LIN {X 0,Y 438.796,Z 820.121,A -85,B 0,C 180,E1 6106.016,E2 6106.016} C_VEL
LIN {X 0,Y 435.592,Z 843.834,A -85,B 0,C 180,E1 6105.62,E2 6105.62} C_VEL
LIN {X 0,Y 431.491,Z 865.928,A -85,B 0,C 180,E1 6105.195,E2 6105.195} C_VEL
LIN {X 0,Y 425.589,Z 891.228,A -85,B 0,C 180,E1 6104.584,E2 6104.584} C_VEL
LIN {X 0,Y 418.146,Z 916.547,A -85,B 0,C 180,E1 6103.788,E2 6103.788} C_VEL
LIN {X 0,Y 411.227,Z 936.788,A -85,B 0,C 180,E1 6103.015,E2 6103.015} C_VEL
LIN {X 0,Y 403.474,Z 956.852,A -85,B 0,C 180,E1 6102.103,E2 6102.103} C_VEL
LIN {X 0,Y 393.277,Z 980.389,A -85,B 0,C 180,E1 6100.823,E2 6100.823} C_VEL
LIN {X 0,Y 381.687,Z 1003.698,A -85,B 0,C 180,E1 6099.261,E2 6099.261} C_VEL
LIN {X 0,Y 371.951,Z 1021.583,A -85,B 0,C 180,E1 6097.831,E2 6097.831} C_VEL
LIN {X 0,Y 361.684,Z 1038.996,A -85,B 0,C 180,E1 6096.212,E2 6096.212} C_VEL
LIN {X 0,Y 348.484,Z 1059.817,A -85,B 0,C 180,E1 6093.904,E2 6093.904} C_VEL
LIN {X 0,Y 335.22,Z 1078.877,A -85,B 0,C 180,E1 6091.299,E2 6091.299} C_VEL
LIN {X 0,Y 323.717,Z 1094.534,A -85,B 0,C 180,E1 6088.74,E2 6088.74} C_VEL
LIN {X 0,Y 310.823,Z 1111.367,A -85,B 0,C 180,E1 6085.438,E2 6085.438} C_VEL
LIN {X 0,Y 298.275,Z 1126.865,A -85,B 0,C 180,E1 6081.666,E2 6081.666} C_VEL
LIN {X 0,Y 288.449,Z 1138.762,A -85,B 0,C 180,E1 6078.182,E2 6078.182} C_VEL
LIN {X 0,Y 279.204,Z 1149.91,A -85,B 0,C 180,E1 6074.292,E2 6074.292} C_VEL
LIN {X 0,Y 269.366,Z 1162.072,A -85,B 0,C 180,E1 6069.121,E2 6069.121} C_VEL
LIN {X 0,Y 261.736,Z 1171.778,A -85,B 0,C 180,E1 6063.899,E2 6063.899} C_VEL
LIN {X 0,Y 256.571,Z 1179.002,A -85,B 0,C 180,E1 6059.152,E2 6059.152} C_VEL
LIN {X 0,Y 252.751,Z 1185.047,A -85,B 0,C 180,E1 6054.294,E2 6054.294} C_VEL
LIN {X 0,Y 249.904,Z 1190.603,A -85,B 0,C 180,E1 6048.667,E2 6048.667} C_VEL
LIN {X 0,Y 248.427,Z 1194.755,A -85,B 0,C 180,E1 6042.789,E2 6042.789} C_VEL
LIN {X 0,Y 248.033,Z 1197.119,A -85,B 0,C 180,E1 6037.644,E2 6037.644} C_VEL
LIN {X 0,Y 247.993,Z 1198.227,A -85,B 0,C 180,E1 6033.235,E2 6033.235} C_VEL
LIN {X 0,Y 248.003,Z 1198.443,A -85,B 0,C 180,E1 6028.844,E2 6028.844} C_VEL
LIN {X 0,Y 247.993,Z 1197.691,A -85,B 0,C 180,E1 6024.214,E2 6024.214} C_VEL
LIN {X 0,Y 248.182,Z 1195.889,A -85,B 0,C 180,E1 6019.435,E2 6019.435} C_VEL
LIN {X 0,Y 248.942,Z 1193.015,A -85,B 0,C 180,E1 6014.575,E2 6014.575} C_VEL
LIN {X 0,Y 250.577,Z 1189.058,A -85,B 0,C 180,E1 6009.686,E2 6009.686} C_VEL
LIN {X 0,Y 253.211,Z 1184.216,A -85,B 0,C 180,E1 6005.006,E2 6005.006} C_VEL
LIN {X 0,Y 257.322,Z 1177.869,A -85,B 0,C 180,E1 6000.058,E2 6000.058} C_VEL
LIN {X 0,Y 264.391,Z 1168.312,A -85,B 0,C 180,E1 5994.113,E2 5994.113} C_VEL
LIN {X 0,Y 272.385,Z 1158.147,A -85,B 0,C 180,E1 5989.131,E2 5989.131} C_VEL
LIN {X 0,Y 280.522,Z 1148.247,A -85,B 0,C 180,E1 5985.11,E2 5985.11} C_VEL
LIN {X 0,Y 290.427,Z 1136.32,A -85,B 0,C 180,E1 5981.064,E2 5981.064} C_VEL
LIN {X 0,Y 303.233,Z 1120.644,A -85,B 0,C 180,E1 5976.748,E2 5976.748} C_VEL
LIN {X 0,Y 314.417,Z 1106.504,A -85,B 0,C 180,E1 5973.572,E2 5973.572} C_VEL
LIN {X 0,Y 325.807,Z 1091.588,A -85,B 0,C 180,E1 5970.762,E2 5970.762} C_VEL
LIN {X 0,Y 339.632,Z 1072.555,A -85,B 0,C 180,E1 5967.788,E2 5967.788} C_VEL
LIN {X 0,Y 352.367,Z 1053.518,A -85,B 0,C 180,E1 5965.371,E2 5965.371} C_VEL
LIN {X 0,Y 363.194,Z 1036.239,A -85,B 0,C 180,E1 5963.528,E2 5963.528} C_VEL
LIN {X 0,Y 374.64,Z 1016.568,A -85,B 0,C 180,E1 5961.754,E2 5961.754} C_VEL
LIN {X 0,Y 386.839,Z 993.292,A -85,B 0,C 180,E1 5960.023,E2 5960.023} C_VEL
LIN {X 0,Y 396.09,Z 973.641,A -85,B 0,C 180,E1 5958.801,E2 5958.801} C_VEL
LIN {X 0,Y 404.283,Z 954.413,A -85,B 0,C 180,E1 5957.788,E2 5957.788} C_VEL
LIN {X 0,Y 412.183,Z 933.675,A -85,B 0,C 180,E1 5956.866,E2 5956.866} C_VEL
LIN {X 0,Y 421.033,Z 906.617,A -85,B 0,C 180,E1 5955.886,E2 5955.886} C_VEL
LIN {X 0,Y 427.259,Z 883.572,A -85,B 0,C 180,E1 5955.226,E2 5955.226} C_VEL
LIN {X 0,Y 432.073,Z 862.129,A -85,B 0,C 180,E1 5954.733,E2 5954.733} C_VEL
LIN {X 0,Y 436.664,Z 836.034,A -85,B 0,C 180,E1 5954.249,E2 5954.249} C_VEL
LIN {X 0,Y 441.088,Z 795.407,A -85,B 0,C 180,E1 5953.614,E2 5953.614} C_VEL
LIN {X 0,Y 460.609,Z 598.366,A -85,B 0,C 180,E1 5950.681,E2 5950.681} C_VEL
LIN {X 0,Y 457.6,Z 592.689,A -85,B 0,C 180,E1 5948.418,E2 5948.418} C_VEL
LIN {X 0,Y 455.635,Z 589.003,A -85,B 0,C 180,E1 5946.616,E2 5946.616} C_VEL
LIN {X 0,Y 454.128,Z 586.275,A -85,B 0,C 180,E1 5944.926,E2 5944.926} C_VEL
LIN {X 0,Y 452.252,Z 582.816,A -85,B 0,C 180,E1 5941.901,E2 5941.901} C_VEL
LIN {X 0,Y 451.266,Z 582.034,A -85,B 0,C 180,E1 5938.222,E2 5938.222} C_VEL
LIN {X 0,Y 451.505,Z 582.728,A -85,B 0,C 180,E1 5935.682,E2 5935.682} C_VEL
LIN {X 0,Y 453.105,Z 586.957,A -85,B 0,C 180,E1 5931.945,E2 5931.945} C_VEL
LIN {X 0,Y 454.885,Z 591.279,A -85,B 0,C 180,E1 5929.616,E2 5929.616} C_VEL
LIN {X 0,Y 457.288,Z 596.631,A -85,B 0,C 180,E1 5927.306,E2 5927.306} C_VEL
LIN {X 0,Y 459.279,Z 601.556,A -85,B 0,C 180,E1 5925.696,E2 5925.696} C_VEL
LIN {X 0,Y 437.308,Z 826.32,A -85,B 0,C 180,E1 5922.449,E2 5922.449} C_VEL
LIN {X 0,Y 434.141,Z 848.783,A -85,B 0,C 180,E1 5922.078,E2 5922.078} C_VEL
LIN {X 0,Y 428.807,Z 875.909,A -85,B 0,C 180,E1 5921.533,E2 5921.533} C_VEL
LIN {X 0,Y 422.894,Z 898.914,A -85,B 0,C 180,E1 5920.937,E2 5920.937} C_VEL
LIN {X 0,Y 416.442,Z 920.116,A -85,B 0,C 180,E1 5920.253,E2 5920.253} C_VEL
LIN {X 0,Y 408.237,Z 943.42,A -85,B 0,C 180,E1 5919.329,E2 5919.329} C_VEL
LIN {X 0,Y 398.118,Z 967.799,A -85,B 0,C 180,E1 5918.126,E2 5918.126} C_VEL
LIN {X 0,Y 389.491,Z 986.265,A -85,B 0,C 180,E1 5917.032,E2 5917.032} C_VEL
LIN {X 0,Y 379.607,Z 1005.443,A -85,B 0,C 180,E1 5915.694,E2 5915.694} C_VEL
LIN {X 0,Y 366.696,Z 1028.066,A -85,B 0,C 180,E1 5913.779,E2 5913.779} C_VEL
LIN {X 0,Y 355.286,Z 1046.089,A -85,B 0,C 180,E1 5911.919,E2 5911.919} C_VEL
LIN {X 0,Y 344.633,Z 1061.765,A -85,B 0,C 180,E1 5910.001,E2 5910.001} C_VEL
LIN {X 0,Y 332.718,Z 1078.203,A -85,B 0,C 180,E1 5907.614,E2 5907.614} C_VEL
LIN {X 0,Y 318.568,Z 1096.284,A -85,B 0,C 180,E1 5904.382,E2 5904.382} C_VEL
LIN {X 0,Y 307.782,Z 1109.336,A -85,B 0,C 180,E1 5901.53,E2 5901.53} C_VEL
LIN {X 0,Y 297.229,Z 1121.639,A -85,B 0,C 180,E1 5898.315,E2 5898.315} C_VEL
LIN {X 0,Y 284.778,Z 1135.724,A -85,B 0,C 180,E1 5893.764,E2 5893.764} C_VEL
LIN {X 0,Y 275.658,Z 1145.826,A -85,B 0,C 180,E1 5889.673,E2 5889.673} C_VEL
LIN {X 0,Y 268.203,Z 1154.193,A -85,B 0,C 180,E1 5885.562,E2 5885.562} C_VEL
LIN {X 0,Y 260.633,Z 1163.104,A -85,B 0,C 180,E1 5880.17,E2 5880.17} C_VEL
LIN {X 0,Y 254.816,Z 1170.36,A -85,B 0,C 180,E1 5874.332,E2 5874.332} C_VEL
LIN {X 0,Y 251.596,Z 1175.02,A -85,B 0,C 180,E1 5869.502,E2 5869.502} C_VEL
LIN {X 0,Y 249.485,Z 1178.756,A -85,B 0,C 180,E1 5864.388,E2 5864.388} C_VEL
LIN {X 0,Y 248.338,Z 1181.722,A -85,B 0,C 180,E1 5858.335,E2 5858.335} C_VEL
LIN {X 0,Y 248.049,Z 1182.949,A -85,B 0,C 180,E1 5853.004,E2 5853.004} C_VEL
LIN {X 0,Y 248.038,Z 1183.109,A -85,B 0,C 180,E1 5848.615,E2 5848.615} C_VEL
LIN {X 0,Y 248.144,Z 1182.396,A -85,B 0,C 180,E1 5843.987,E2 5843.987} C_VEL
LIN {X 0,Y 248.625,Z 1180.776,A -85,B 0,C 180,E1 5839.34,E2 5839.34} C_VEL
LIN {X 0,Y 249.756,Z 1178.231,A -85,B 0,C 180,E1 5834.68,E2 5834.68} C_VEL
LIN {X 0,Y 251.931,Z 1174.534,A -85,B 0,C 180,E1 5829.801,E2 5829.801} C_VEL
LIN {X 0,Y 256.315,Z 1168.527,A -85,B 0,C 180,E1 5823.845,E2 5823.845} C_VEL
LIN {X 0,Y 262.455,Z 1160.894,A -85,B 0,C 180,E1 5818.283,E2 5818.283} C_VEL
LIN {X 0,Y 269.126,Z 1153.218,A -85,B 0,C 180,E1 5813.792,E2 5813.792} C_VEL
LIN {X 0,Y 278.439,Z 1142.928,A -85,B 0,C 180,E1 5808.917,E2 5808.917} C_VEL
LIN {X 0,Y 289.405,Z 1130.604,A -85,B 0,C 180,E1 5804.343,E2 5804.343} C_VEL
LIN {X 0,Y 299.489,Z 1119.152,A -85,B 0,C 180,E1 5800.873,E2 5800.873} C_VEL
LIN {X 0,Y 311.744,Z 1104.868,A -85,B 0,C 180,E1 5797.305,E2 5797.305} C_VEL
LIN {X 0,Y 324.711,Z 1088.751,A -85,B 0,C 180,E1 5794.074,E2 5794.074} C_VEL
LIN {X 0,Y 335.895,Z 1074.082,A -85,B 0,C 180,E1 5791.642,E2 5791.642} C_VEL
LIN {X 0,Y 346.923,Z 1058.74,A -85,B 0,C 180,E1 5789.495,E2 5789.495} C_VEL
LIN {X 0,Y 360.604,Z 1038.215,A -85,B 0,C 180,E1 5787.12,E2 5787.12} C_VEL
LIN {X 0,Y 371.794,Z 1019.69,A -85,B 0,C 180,E1 5785.364,E2 5785.364} C_VEL
LIN {X 0,Y 381.756,Z 1001.755,A -85,B 0,C 180,E1 5783.925,E2 5783.925} C_VEL
LIN {X 0,Y 392.363,Z 980.824,A -85,B 0,C 180,E1 5782.517,E2 5782.517} C_VEL
LIN {X 0,Y 403.186,Z 956.416,A -85,B 0,C 180,E1 5781.18,E2 5781.18} C_VEL
LIN {X 0,Y 410.938,Z 936.563,A -85,B 0,C 180,E1 5780.286,E2 5780.286} C_VEL
LIN {X 0,Y 417.942,Z 916.134,A -85,B 0,C 180,E1 5779.508,E2 5779.508} C_VEL
LIN {X 0,Y 425.586,Z 889.88,A -85,B 0,C 180,E1 5778.706,E2 5778.706} C_VEL
LIN {X 0,Y 431.196,Z 865.565,A -85,B 0,C 180,E1 5778.142,E2 5778.142} C_VEL
LIN {X 0,Y 435.188,Z 843.579,A -85,B 0,C 180,E1 5777.734,E2 5777.734} C_VEL
LIN {X 0,Y 436.959,Z 831.119,A -85,B 0,C 180,E1 5777.528,E2 5777.528} C_VEL
LIN {X 0,Y 437.578,Z 823.596,A -85,B 0,C 180,E1 5777.288,E2 5777.288} C_VEL
LIN {X 0,Y 437.97,Z 804.029,A -85,B 0,C 180,E1 5776.203,E2 5776.203} C_VEL
LIN {X 0,Y 438.401,Z 797.543,A -85,B 0,C 180,E1 5776.014,E2 5776.014} C_VEL
LIN {X 0,Y 457.292,Z 607.146,A -85,B 0,C 180,E1 5773.293,E2 5773.293} C_VEL
LIN {X 0,Y 454.572,Z 600.576,A -85,B 0,C 180,E1 5770.776,E2 5770.776} C_VEL
LIN {X 0,Y 452.457,Z 595.594,A -85,B 0,C 180,E1 5768.131,E2 5768.131} C_VEL
LIN {X 0,Y 451.655,Z 593.668,A -85,B 0,C 180,E1 5766.738,E2 5766.738} C_VEL
LIN {X 0,Y 450.659,Z 590.496,A -85,B 0,C 180,E1 5763.434,E2 5763.434} C_VEL
LIN {X 0,Y 450.86,Z 590.358,A -85,B 0,C 180,E1 5759.873,E2 5759.873} C_VEL
LIN {X 0,Y 451.639,Z 591.215,A -85,B 0,C 180,E1 5757.843,E2 5757.843} C_VEL
LIN {X 0,Y 453.942,Z 595.56,A -85,B 0,C 180,E1 5754.375,E2 5754.375} C_VEL
LIN {X 0,Y 456.023,Z 599.584,A -85,B 0,C 180,E1 5752.25,E2 5752.25} C_VEL
LIN {X 0,Y 458.505,Z 604.367,A -85,B 0,C 180,E1 5750.218,E2 5750.218} C_VEL
LIN {X 0,Y 436.503,Z 821.567,A -85,B 0,C 180,E1 5747.007,E2 5747.007} C_VEL
LIN {X 0,Y 433.318,Z 844.483,A -85,B 0,C 180,E1 5746.628,E2 5746.628} C_VEL
LIN {X 0,Y 429.076,Z 866.856,A -85,B 0,C 180,E1 5746.203,E2 5746.203} C_VEL
LIN {X 0,Y 422.777,Z 893.065,A -85,B 0,C 180,E1 5745.574,E2 5745.574} C_VEL
LIN {X 0,Y 415.449,Z 917.389,A -85,B 0,C 180,E1 5744.817,E2 5744.817} C_VEL
LIN {X 0,Y 408.62,Z 937.002,A -85,B 0,C 180,E1 5744.081,E2 5744.081} C_VEL
LIN {X 0,Y 400.598,Z 957.382,A -85,B 0,C 180,E1 5743.17,E2 5743.17} C_VEL
LIN {X 0,Y 389.823,Z 981.671,A -85,B 0,C 180,E1 5741.862,E2 5741.862} C_VEL
LIN {X 0,Y 378.65,Z 1003.647,A -85,B 0,C 180,E1 5740.405,E2 5740.405} C_VEL
LIN {X 0,Y 368.503,Z 1021.888,A -85,B 0,C 180,E1 5738.969,E2 5738.969} C_VEL
LIN {X 0,Y 357.598,Z 1039.945,A -85,B 0,C 180,E1 5737.302,E2 5737.302} C_VEL
LIN {X 0,Y 343.413,Z 1061.561,A -85,B 0,C 180,E1 5734.89,E2 5734.89} C_VEL
LIN {X 0,Y 331.214,Z 1078.635,A -85,B 0,C 180,E1 5732.564,E2 5732.564} C_VEL
LIN {X 0,Y 319.585,Z 1094.023,A -85,B 0,C 180,E1 5730.07,E2 5730.07} C_VEL
LIN {X 0,Y 306.717,Z 1110.28,A -85,B 0,C 180,E1 5726.908,E2 5726.908} C_VEL
LIN {X 0,Y 293.101,Z 1126.583,A -85,B 0,C 180,E1 5722.964,E2 5722.964} C_VEL
LIN {X 0,Y 282.726,Z 1138.66,A -85,B 0,C 180,E1 5719.403,E2 5719.403} C_VEL
LIN {X 0,Y 273.221,Z 1149.634,A -85,B 0,C 180,E1 5715.529,E2 5715.529} C_VEL
LIN {X 0,Y 262.87,Z 1161.797,A -85,B 0,C 180,E1 5710.287,E2 5710.287} C_VEL
LIN {X 0,Y 254.667,Z 1171.673,A -85,B 0,C 180,E1 5704.856,E2 5704.856} C_VEL
LIN {X 0,Y 249.292,Z 1178.739,A -85,B 0,C 180,E1 5700.089,E2 5700.089} C_VEL
LIN {X 0,Y 245.19,Z 1184.787,A -85,B 0,C 180,E1 5695.094,E2 5695.094} C_VEL
LIN {X 0,Y 242.112,Z 1190.347,A -85,B 0,C 180,E1 5689.292,E2 5689.292} C_VEL
LIN {X 0,Y 240.489,Z 1194.504,A -85,B 0,C 180,E1 5683.218,E2 5683.218} C_VEL
LIN {X 0,Y 240.04,Z 1196.87,A -85,B 0,C 180,E1 5677.9,E2 5677.9} C_VEL
LIN {X 0,Y 239.994,Z 1197.98,A -85,B 0,C 180,E1 5673.343,E2 5673.343} C_VEL
LIN {X 0,Y 240.006,Z 1198.196,A -85,B 0,C 180,E1 5668.806,E2 5668.806} C_VEL
LIN {X 0,Y 239.997,Z 1197.442,A -85,B 0,C 180,E1 5664.021,E2 5664.021} C_VEL
LIN {X 0,Y 240.199,Z 1195.698,A -85,B 0,C 180,E1 5659.203,E2 5659.203} C_VEL
LIN {X 0,Y 241.043,Z 1192.797,A -85,B 0,C 180,E1 5654.11,E2 5654.11} C_VEL
LIN {X 0,Y 242.841,Z 1188.8,A -85,B 0,C 180,E1 5649.009,E2 5649.009} C_VEL
LIN {X 0,Y 245.692,Z 1183.955,A -85,B 0,C 180,E1 5644.185,E2 5644.185} C_VEL
LIN {X 0,Y 249.987,Z 1177.748,A -85,B 0,C 180,E1 5639.205,E2 5639.205} C_VEL
LIN {X 0,Y 257.286,Z 1168.461,A -85,B 0,C 180,E1 5633.238,E2 5633.238} C_VEL
LIN {X 0,Y 265.956,Z 1157.992,A -85,B 0,C 180,E1 5627.994,E2 5627.994} C_VEL
LIN {X 0,Y 274.595,Z 1147.97,A -85,B 0,C 180,E1 5623.865,E2 5623.865} C_VEL
LIN {X 0,Y 284.932,Z 1136.038,A -85,B 0,C 180,E1 5619.779,E2 5619.779} C_VEL
LIN {X 0,Y 298.25,Z 1120.349,A -85,B 0,C 180,E1 5615.446,E2 5615.446} C_VEL
LIN {X 0,Y 309.832,Z 1106.204,A -85,B 0,C 180,E1 5612.272,E2 5612.272} C_VEL
LIN {X 0,Y 320.911,Z 1092.143,A -85,B 0,C 180,E1 5609.623,E2 5609.623} C_VEL
LIN {X 0,Y 334.737,Z 1073.742,A -85,B 0,C 180,E1 5606.73,E2 5606.73} C_VEL
LIN {X 0,Y 348.221,Z 1054.156,A -85,B 0,C 180,E1 5604.244,E2 5604.244} C_VEL
LIN {X 0,Y 359.322,Z 1036.885,A -85,B 0,C 180,E1 5602.41,E2 5602.41} C_VEL
LIN {X 0,Y 370.456,Z 1018.221,A -85,B 0,C 180,E1 5600.736,E2 5600.736} C_VEL
LIN {X 0,Y 383.154,Z 994.751,A -85,B 0,C 180,E1 5598.989,E2 5598.989} C_VEL
LIN {X 0,Y 392.996,Z 974.303,A -85,B 0,C 180,E1 5597.729,E2 5597.729} C_VEL
LIN {X 0,Y 401.43,Z 954.907,A -85,B 0,C 180,E1 5596.722,E2 5596.722} C_VEL
LIN {X 0,Y 409.456,Z 934.239,A -85,B 0,C 180,E1 5595.817,E2 5595.817} C_VEL
LIN {X 0,Y 418.228,Z 908.105,A -85,B 0,C 180,E1 5594.881,E2 5594.881} C_VEL
LIN {X 0,Y 424.87,Z 883.989,A -85,B 0,C 180,E1 5594.2,E2 5594.2} C_VEL
LIN {X 0,Y 429.753,Z 862.607,A -85,B 0,C 180,E1 5593.717,E2 5593.717} C_VEL
LIN {X 0,Y 434.19,Z 837.948,A -85,B 0,C 180,E1 5593.265,E2 5593.265} C_VEL
LIN {X 0,Y 438.389,Z 801.607,A -85,B 0,C 180,E1 5592.697,E2 5592.697} C_VEL
LIN {X 0,Y 458.297,Z 604.189,A -85,B 0,C 180,E1 5589.782,E2 5589.782} C_VEL
LIN {X 0,Y 455.023,Z 597.759,A -85,B 0,C 180,E1 5587.005,E2 5587.005} C_VEL
LIN {X 0,Y 453.034,Z 594.148,A -85,B 0,C 180,E1 5584.811,E2 5584.811} C_VEL
LIN {X 0,Y 451.209,Z 590.714,A -85,B 0,C 180,E1 5581.778,E2 5581.778} C_VEL
LIN {X 0,Y 450.286,Z 589.974,A -85,B 0,C 180,E1 5578.218,E2 5578.218} C_VEL
LIN {X 0,Y 450.525,Z 590.758,A -85,B 0,C 180,E1 5575.672,E2 5575.672} C_VEL
LIN {X 0,Y 452.006,Z 594.767,A -85,B 0,C 180,E1 5572.117,E2 5572.117} C_VEL
LIN {X 0,Y 453.731,Z 599.105,A -85,B 0,C 180,E1 5569.782,E2 5569.782} C_VEL
LIN {X 0,Y 456.149,Z 604.706,A -85,B 0,C 180,E1 5567.402,E2 5567.402} C_VEL
LIN {X 0,Y 457.073,Z 607.226,A -85,B 0,C 180,E1 5566.599,E2 5566.599} C_VEL
LIN {X 0,Y 435.048,Z 827.651,A -85,B 0,C 180,E1 5563.446,E2 5563.446} C_VEL
LIN {X 0,Y 431.48,Z 851.887,A -85,B 0,C 180,E1 5563.048,E2 5563.048} C_VEL
LIN {X 0,Y 425.687,Z 879.45,A -85,B 0,C 180,E1 5562.485,E2 5562.485} C_VEL
LIN {X 0,Y 420.148,Z 900.383,A -85,B 0,C 180,E1 5561.942,E2 5561.942} C_VEL
LIN {X 0,Y 413.814,Z 920.754,A -85,B 0,C 180,E1 5561.294,E2 5561.294} C_VEL
LIN {X 0,Y 405.067,Z 945.091,A -85,B 0,C 180,E1 5560.34,E2 5560.34} C_VEL
LIN {X 0,Y 395.195,Z 968.26,A -85,B 0,C 180,E1 5559.207,E2 5559.207} C_VEL
LIN {X 0,Y 386.266,Z 986.989,A -85,B 0,C 180,E1 5558.114,E2 5558.114} C_VEL
LIN {X 0,Y 375.96,Z 1006.562,A -85,B 0,C 180,E1 5556.762,E2 5556.762} C_VEL
LIN {X 0,Y 362.417,Z 1029.615,A -85,B 0,C 180,E1 5554.814,E2 5554.814} C_VEL
LIN {X 0,Y 351.157,Z 1046.969,A -85,B 0,C 180,E1 5553.029,E2 5553.029} C_VEL
LIN {X 0,Y 339.838,Z 1063.18,A -85,B 0,C 180,E1 5551.047,E2 5551.047} C_VEL
LIN {X 0,Y 325.684,Z 1082.015,A -85,B 0,C 180,E1 5548.257,E2 5548.257} C_VEL
LIN {X 0,Y 313.213,Z 1097.329,A -85,B 0,C 180,E1 5545.449,E2 5545.449} C_VEL
LIN {X 0,Y 302.128,Z 1110.305,A -85,B 0,C 180,E1 5542.587,E2 5542.587} C_VEL
LIN {X 0,Y 290.168,Z 1123.778,A -85,B 0,C 180,E1 5538.995,E2 5538.995} C_VEL
LIN {X 0,Y 277.901,Z 1136.994,A -85,B 0,C 180,E1 5534.556,E2 5534.556} C_VEL
LIN {X 0,Y 268.925,Z 1146.538,A -85,B 0,C 180,E1 5530.592,E2 5530.592} C_VEL
LIN {X 0,Y 260.812,Z 1155.24,A -85,B 0,C 180,E1 5526.185,E2 5526.185} C_VEL
LIN {X 0,Y 252.439,Z 1164.551,A -85,B 0,C 180,E1 5520.201,E2 5520.201} C_VEL
LIN {X 0,Y 247.16,Z 1170.861,A -85,B 0,C 180,E1 5514.881,E2 5514.881} C_VEL
LIN {X 0,Y 243.774,Z 1175.472,A -85,B 0,C 180,E1 5509.904,E2 5509.904} C_VEL
LIN {X 0,Y 241.45,Z 1179.371,A -85,B 0,C 180,E1 5504.294,E2 5504.294} C_VEL
LIN {X 0,Y 240.319,Z 1182.098,A -85,B 0,C 180,E1 5498.133,E2 5498.133} C_VEL
LIN {X 0,Y 240.054,Z 1183.196,A -85,B 0,C 180,E1 5493.104,E2 5493.104} C_VEL
LIN {X 0,Y 240.041,Z 1183.356,A -85,B 0,C 180,E1 5488.568,E2 5488.568} C_VEL
LIN {X 0,Y 240.16,Z 1182.644,A -85,B 0,C 180,E1 5483.786,E2 5483.786} C_VEL
LIN {X 0,Y 240.647,Z 1181.134,A -85,B 0,C 180,E1 5479.224,E2 5479.224} C_VEL
LIN {X 0,Y 241.919,Z 1178.482,A -85,B 0,C 180,E1 5474.171,E2 5474.171} C_VEL
LIN {X 0,Y 244.264,Z 1174.786,A -85,B 0,C 180,E1 5469.138,E2 5469.138} C_VEL
LIN {X 0,Y 248.838,Z 1168.92,A -85,B 0,C 180,E1 5463.132,E2 5463.132} C_VEL
LIN {X 0,Y 255.488,Z 1161.128,A -85,B 0,C 180,E1 5457.292,E2 5457.292} C_VEL
LIN {X 0,Y 262.5,Z 1153.477,A -85,B 0,C 180,E1 5452.726,E2 5452.726} C_VEL
LIN {X 0,Y 271.811,Z 1143.635,A -85,B 0,C 180,E1 5447.972,E2 5447.972} C_VEL
LIN {X 0,Y 283.18,Z 1131.432,A -85,B 0,C 180,E1 5443.335,E2 5443.335} C_VEL
LIN {X 0,Y 293.876,Z 1119.731,A -85,B 0,C 180,E1 5439.742,E2 5439.742} C_VEL
LIN {X 0,Y 304.982,Z 1107.202,A -85,B 0,C 180,E1 5436.561,E2 5436.561} C_VEL
LIN {X 0,Y 319.647,Z 1089.718,A -85,B 0,C 180,E1 5432.976,E2 5432.976} C_VEL
LIN {X 0,Y 330.981,Z 1075.293,A -85,B 0,C 180,E1 5430.575,E2 5430.575} C_VEL
LIN {X 0,Y 341.93,Z 1060.496,A -85,B 0,C 180,E1 5428.494,E2 5428.494} C_VEL
LIN {X 0,Y 353.969,Z 1043.092,A -85,B 0,C 180,E1 5426.435,E2 5426.435} C_VEL
LIN {X 0,Y 367.623,Z 1021.367,A -85,B 0,C 180,E1 5424.337,E2 5424.337} C_VEL
LIN {X 0,Y 377.967,Z 1003.21,A -85,B 0,C 180,E1 5422.885,E2 5422.885} C_VEL
LIN {X 0,Y 387.734,Z 984.447,A -85,B 0,C 180,E1 5421.621,E2 5421.621} C_VEL
LIN {X 0,Y 398.725,Z 960.887,A -85,B 0,C 180,E1 5420.304,E2 5420.304} C_VEL
LIN {X 0,Y 407.816,Z 938.233,A -85,B 0,C 180,E1 5419.277,E2 5419.277} C_VEL
LIN {X 0,Y 414.921,Z 918.031,A -85,B 0,C 180,E1 5418.513,E2 5418.513} C_VEL
LIN {X 0,Y 421.939,Z 894.911,A -85,B 0,C 180,E1 5417.8,E2 5417.8} C_VEL
LIN {X 0,Y 428.578,Z 867.625,A -85,B 0,C 180,E1 5417.156,E2 5417.156} C_VEL
LIN {X 0,Y 432.761,Z 845.353,A -85,B 0,C 180,E1 5416.743,E2 5416.743} C_VEL
LIN {X 0,Y 435.945,Z 821.931,A -85,B 0,C 180,E1 5416.369,E2 5416.369} C_VEL
LIN {X 0,Y 438.401,Z 797.543,A -85,B 0,C 180,E1 5416.014,E2 5416.014} C_VEL
LIN {X 0,Y 438.892,Z 790.003,A -85,B 0,C 180,E1 5415.78,E2 5415.78} C_VEL
LIN {X 0,Y 439.359,Z 770.428,A -85,B 0,C 180,E1 5414.702,E2 5414.702} C_VEL
LIN {X 0,Y 439.841,Z 763.942,A -85,B 0,C 180,E1 5414.516,E2 5414.516} C_VEL
LIN {X 0,Y 455.199,Z 612.867,A -85,B 0,C 180,E1 5412.383,E2 5412.383} C_VEL
LIN {X 0,Y 452.836,Z 607.181,A -85,B 0,C 180,E1 5409.982,E2 5409.982} C_VEL
LIN {X 0,Y 451.17,Z 602.87,A -85,B 0,C 180,E1 5407.641,E2 5407.641} C_VEL
LIN {X 0,Y 450.237,Z 600.725,A -85,B 0,C 180,E1 5405.787,E2 5405.787} C_VEL
LIN {X 0,Y 449.679,Z 598.441,A -85,B 0,C 180,E1 5403.442,E2 5403.442} C_VEL
LIN {X 0,Y 449.878,Z 598.3,A -85,B 0,C 180,E1 5399.873,E2 5399.873} C_VEL
LIN {X 0,Y 450.647,Z 599.257,A -85,B 0,C 180,E1 5397.838,E2 5397.838} C_VEL
LIN {X 0,Y 452.779,Z 603.355,A -85,B 0,C 180,E1 5394.551,E2 5394.551} C_VEL
LIN {X 0,Y 454.74,Z 607.263,A -85,B 0,C 180,E1 5392.482,E2 5392.482} C_VEL
LIN {X 0,Y 456.293,Z 610.506,A -85,B 0,C 180,E1 5391.114,E2 5391.114} C_VEL
LIN {X 0,Y 434.186,Z 824.271,A -85,B 0,C 180,E1 5387.988,E2 5387.988} C_VEL
LIN {X 0,Y 430.933,Z 846.6,A -85,B 0,C 180,E1 5387.621,E2 5387.621} C_VEL
LIN {X 0,Y 425.667,Z 873.141,A -85,B 0,C 180,E1 5387.114,E2 5387.114} C_VEL
LIN {X 0,Y 419.035,Z 898.394,A -85,B 0,C 180,E1 5386.476,E2 5386.476} C_VEL
LIN {X 0,Y 412.514,Z 919.346,A -85,B 0,C 180,E1 5385.822,E2 5385.822} C_VEL
LIN {X 0,Y 405.159,Z 939.866,A -85,B 0,C 180,E1 5385.052,E2 5385.052} C_VEL
LIN {X 0,Y 395.344,Z 963.949,A -85,B 0,C 180,E1 5383.959,E2 5383.959} C_VEL
LIN {X 0,Y 384.408,Z 987.004,A -85,B 0,C 180,E1 5382.667,E2 5382.667} C_VEL
LIN {X 0,Y 374.507,Z 1005.884,A -85,B 0,C 180,E1 5381.404,E2 5381.404} C_VEL
LIN {X 0,Y 364.006,Z 1024.227,A -85,B 0,C 180,E1 5379.955,E2 5379.955} C_VEL
LIN {X 0,Y 350.636,Z 1045.616,A -85,B 0,C 180,E1 5377.936,E2 5377.936} C_VEL
LIN {X 0,Y 337.702,Z 1064.338,A -85,B 0,C 180,E1 5375.773,E2 5375.773} C_VEL
LIN {X 0,Y 325.994,Z 1080.211,A -85,B 0,C 180,E1 5373.586,E2 5373.586} C_VEL
LIN {X 0,Y 313.862,Z 1095.753,A -85,B 0,C 180,E1 5371.037,E2 5371.037} C_VEL
LIN {X 0,Y 298.393,Z 1114.433,A -85,B 0,C 180,E1 5367.252,E2 5367.252} C_VEL
LIN {X 0,Y 286.736,Z 1127.81,A -85,B 0,C 180,E1 5363.891,E2 5363.891} C_VEL
LIN {X 0,Y 276.389,Z 1139.387,A -85,B 0,C 180,E1 5360.403,E2 5360.403} C_VEL
LIN {X 0,Y 265.024,Z 1152.015,A -85,B 0,C 180,E1 5355.793,E2 5355.793} C_VEL
LIN {X 0,Y 254.412,Z 1163.785,A -85,B 0,C 180,E1 5350.318,E2 5350.318} C_VEL
LIN {X 0,Y 247.32,Z 1171.984,A -85,B 0,C 180,E1 5345.603,E2 5345.603} C_VEL
LIN {X 0,Y 241.582,Z 1179.133,A -85,B 0,C 180,E1 5340.582,E2 5340.582} C_VEL
LIN {X 0,Y 236.537,Z 1186.386,A -85,B 0,C 180,E1 5334.206,E2 5334.206} C_VEL
LIN {X 0,Y 233.536,Z 1191.719,A -85,B 0,C 180,E1 5327.696,E2 5327.696} C_VEL
LIN {X 0,Y 232.401,Z 1194.737,A -85,B 0,C 180,E1 5322.675,E2 5322.675} C_VEL
LIN {X 0,Y 232.042,Z 1196.694,A -85,B 0,C 180,E1 5317.925,E2 5317.925} C_VEL
LIN {X 0,Y 231.997,Z 1197.733,A -85,B 0,C 180,E1 5313.459,E2 5313.459} C_VEL
LIN {X 0,Y 232.01,Z 1197.949,A -85,B 0,C 180,E1 5308.765,E2 5308.765} C_VEL
LIN {X 0,Y 231.999,Z 1197.266,A -85,B 0,C 180,E1 5304.062,E2 5304.062} C_VEL
LIN {X 0,Y 232.231,Z 1195.447,A -85,B 0,C 180,E1 5298.828,E2 5298.828} C_VEL
LIN {X 0,Y 233.171,Z 1192.542,A -85,B 0,C 180,E1 5293.559,E2 5293.559} C_VEL
LIN {X 0,Y 235.013,Z 1188.759,A -85,B 0,C 180,E1 5288.537,E2 5288.537} C_VEL
LIN {X 0,Y 238.135,Z 1183.816,A -85,B 0,C 180,E1 5283.426,E2 5283.426} C_VEL
LIN {X 0,Y 242.824,Z 1177.483,A -85,B 0,C 180,E1 5278.192,E2 5278.192} C_VEL
LIN {X 0,Y 250.578,Z 1168.19,A -85,B 0,C 180,E1 5272.084,E2 5272.084} C_VEL
LIN {X 0,Y 259.744,Z 1157.72,A -85,B 0,C 180,E1 5266.748,E2 5266.748} C_VEL
LIN {X 0,Y 268.795,Z 1147.692,A -85,B 0,C 180,E1 5262.563,E2 5262.563} C_VEL
LIN {X 0,Y 279.587,Z 1135.757,A -85,B 0,C 180,E1 5258.445,E2 5258.445} C_VEL
LIN {X 0,Y 293.431,Z 1120.057,A -85,B 0,C 180,E1 5254.102,E2 5254.102} C_VEL
LIN {X 0,Y 305.454,Z 1105.858,A -85,B 0,C 180,E1 5250.926,E2 5250.926} C_VEL
LIN {X 0,Y 317.244,Z 1091.333,A -85,B 0,C 180,E1 5248.214,E2 5248.214} C_VEL
LIN {X 0,Y 331.784,Z 1072.408,A -85,B 0,C 180,E1 5245.298,E2 5245.298} C_VEL
LIN {X 0,Y 345.223,Z 1053.302,A -85,B 0,C 180,E1 5242.922,E2 5242.922} C_VEL
LIN {X 0,Y 356.404,Z 1036.248,A -85,B 0,C 180,E1 5241.145,E2 5241.145} C_VEL
LIN {X 0,Y 368,Z 1017.161,A -85,B 0,C 180,E1 5239.469,E2 5239.469} C_VEL
LIN {X 0,Y 381.357,Z 992.687,A -85,B 0,C 180,E1 5237.707,E2 5237.707} C_VEL
LIN {X 0,Y 391.092,Z 972.689,A -85,B 0,C 180,E1 5236.516,E2 5236.516} C_VEL
LIN {X 0,Y 399.957,Z 952.453,A -85,B 0,C 180,E1 5235.504,E2 5235.504} C_VEL
LIN {X 0,Y 409.468,Z 927.866,A -85,B 0,C 180,E1 5234.485,E2 5234.485} C_VEL
LIN {X 0,Y 417.491,Z 902.953,A -85,B 0,C 180,E1 5233.664,E2 5233.664} C_VEL
LIN {X 0,Y 423.297,Z 881.701,A -85,B 0,C 180,E1 5233.096,E2 5233.096} C_VEL
LIN {X 0,Y 428.466,Z 858.843,A -85,B 0,C 180,E1 5232.606,E2 5232.606} C_VEL
LIN {X 0,Y 433.337,Z 829.443,A -85,B 0,C 180,E1 5232.1,E2 5232.1} C_VEL
LIN {X 0,Y 441.651,Z 750.287,A -85,B 0,C 180,E1 5230.922,E2 5230.922} C_VEL
LIN {X 0,Y 456.066,Z 610.091,A -85,B 0,C 180,E1 5228.86,E2 5228.86} C_VEL
LIN {X 0,Y 453.394,Z 604.808,A -85,B 0,C 180,E1 5226.394,E2 5226.394} C_VEL
LIN {X 0,Y 451.846,Z 601.877,A -85,B 0,C 180,E1 5224.569,E2 5224.569} C_VEL
LIN {X 0,Y 450.171,Z 598.611,A -85,B 0,C 180,E1 5221.655,E2 5221.655} C_VEL
LIN {X 0,Y 449.303,Z 597.927,A -85,B 0,C 180,E1 5218.087,E2 5218.087} C_VEL
LIN {X 0,Y 449.524,Z 598.643,A -85,B 0,C 180,E1 5215.791,E2 5215.791} C_VEL
LIN {X 0,Y 450.944,Z 602.686,A -85,B 0,C 180,E1 5212.226,E2 5212.226} C_VEL
LIN {X 0,Y 452.804,Z 607.432,A -85,B 0,C 180,E1 5209.696,E2 5209.696} C_VEL
LIN {X 0,Y 454.999,Z 612.74,A -85,B 0,C 180,E1 5207.512,E2 5207.512} C_VEL
LIN {X 0,Y 433.009,Z 828.267,A -85,B 0,C 180,E1 5204.464,E2 5204.464} C_VEL
LIN {X 0,Y 429.022,Z 854.51,A -85,B 0,C 180,E1 5204.037,E2 5204.037} C_VEL
LIN {X 0,Y 423.252,Z 880.748,A -85,B 0,C 180,E1 5203.502,E2 5203.502} C_VEL
LIN {X 0,Y 417.746,Z 901.117,A -85,B 0,C 180,E1 5202.981,E2 5202.981} C_VEL
LIN {X 0,Y 410.897,Z 922.667,A -85,B 0,C 180,E1 5202.303,E2 5202.303} C_VEL
LIN {X 0,Y 400.708,Z 949.694,A -85,B 0,C 180,E1 5201.233,E2 5201.233} C_VEL
LIN {X 0,Y 392,Z 969.611,A -85,B 0,C 180,E1 5200.257,E2 5200.257} C_VEL
LIN {X 0,Y 382.953,Z 988.165,A -85,B 0,C 180,E1 5199.185,E2 5199.185} C_VEL
LIN {X 0,Y 371.166,Z 1010.02,A -85,B 0,C 180,E1 5197.676,E2 5197.676} C_VEL
LIN {X 0,Y 358.26,Z 1031.161,A -85,B 0,C 180,E1 5195.872,E2 5195.872} C_VEL
LIN {X 0,Y 347.163,Z 1047.847,A -85,B 0,C 180,E1 5194.164,E2 5194.164} C_VEL
LIN {X 0,Y 334.942,Z 1064.895,A -85,B 0,C 180,E1 5192.084,E2 5192.084} C_VEL
LIN {X 0,Y 319.666,Z 1084.439,A -85,B 0,C 180,E1 5189.137,E2 5189.137} C_VEL
LIN {X 0,Y 307.971,Z 1098.371,A -85,B 0,C 180,E1 5186.553,E2 5186.553} C_VEL
LIN {X 0,Y 296.582,Z 1111.272,A -85,B 0,C 180,E1 5183.683,E2 5183.683} C_VEL
LIN {X 0,Y 283.144,Z 1125.842,A -85,B 0,C 180,E1 5179.709,E2 5179.709} C_VEL
LIN {X 0,Y 271.573,Z 1137.762,A -85,B 0,C 180,E1 5175.584,E2 5175.584} C_VEL
LIN {X 0,Y 262.264,Z 1147.248,A -85,B 0,C 180,E1 5171.558,E2 5171.558} C_VEL
LIN {X 0,Y 253.093,Z 1156.681,A -85,B 0,C 180,E1 5166.624,E2 5166.624} C_VEL
LIN {X 0,Y 244.786,Z 1165.391,A -85,B 0,C 180,E1 5160.703,E2 5160.703} C_VEL
LIN {X 0,Y 239.526,Z 1171.36,A -85,B 0,C 180,E1 5155.466,E2 5155.466} C_VEL
LIN {X 0,Y 235.827,Z 1176.12,A -85,B 0,C 180,E1 5150.087,E2 5150.087} C_VEL
LIN {X 0,Y 233.196,Z 1180.361,A -85,B 0,C 180,E1 5143.388,E2 5143.388} C_VEL
LIN {X 0,Y 232.3,Z 1182.474,A -85,B 0,C 180,E1 5137.917,E2 5137.917} C_VEL
LIN {X 0,Y 232.055,Z 1183.464,A -85,B 0,C 180,E1 5132.964,E2 5132.964} C_VEL
LIN {X 0,Y 232.045,Z 1183.603,A -85,B 0,C 180,E1 5128.519,E2 5128.519} C_VEL
LIN {X 0,Y 232.178,Z 1182.892,A -85,B 0,C 180,E1 5123.572,E2 5123.572} C_VEL
LIN {X 0,Y 232.708,Z 1181.383,A -85,B 0,C 180,E1 5118.852,E2 5118.852} C_VEL
LIN {X 0,Y 234.101,Z 1178.733,A -85,B 0,C 180,E1 5113.627,E2 5113.627} C_VEL
LIN {X 0,Y 236.689,Z 1174.966,A -85,B 0,C 180,E1 5108.34,E2 5108.34} C_VEL
LIN {X 0,Y 241.646,Z 1169.039,A -85,B 0,C 180,E1 5102.124,E2 5102.124} C_VEL
LIN {X 0,Y 248.552,Z 1161.41,A -85,B 0,C 180,E1 5096.28,E2 5096.28} C_VEL
LIN {X 0,Y 255.97,Z 1153.736,A -85,B 0,C 180,E1 5091.605,E2 5091.605} C_VEL
LIN {X 0,Y 265.721,Z 1143.896,A -85,B 0,C 180,E1 5086.777,E2 5086.777} C_VEL
LIN {X 0,Y 277.724,Z 1131.542,A -85,B 0,C 180,E1 5082.041,E2 5082.041} C_VEL
LIN {X 0,Y 288.67,Z 1120.001,A -85,B 0,C 180,E1 5078.483,E2 5078.483} C_VEL
LIN {X 0,Y 300.149,Z 1107.478,A -85,B 0,C 180,E1 5075.298,E2 5075.298} C_VEL
LIN {X 0,Y 315.125,Z 1090.163,A -85,B 0,C 180,E1 5071.751,E2 5071.751} C_VEL
LIN {X 0,Y 327.597,Z 1074.682,A -85,B 0,C 180,E1 5069.201,E2 5069.201} C_VEL
LIN {X 0,Y 338.814,Z 1059.857,A -85,B 0,C 180,E1 5067.158,E2 5067.158} C_VEL
LIN {X 0,Y 351.958,Z 1041.225,A -85,B 0,C 180,E1 5065.009,E2 5065.009} C_VEL
LIN {X 0,Y 365.147,Z 1020.409,A -85,B 0,C 180,E1 5063.066,E2 5063.066} C_VEL
LIN {X 0,Y 375.494,Z 1002.521,A -85,B 0,C 180,E1 5061.671,E2 5061.671} C_VEL
LIN {X 0,Y 385.657,Z 983.253,A -85,B 0,C 180,E1 5060.407,E2 5060.407} C_VEL
LIN {X 0,Y 397.668,Z 957.404,A -85,B 0,C 180,E1 5059.023,E2 5059.023} C_VEL
LIN {X 0,Y 405.667,Z 937.662,A -85,B 0,C 180,E1 5058.165,E2 5058.165} C_VEL
LIN {X 0,Y 412.456,Z 918.65,A -85,B 0,C 180,E1 5057.462,E2 5057.462} C_VEL
LIN {X 0,Y 419.126,Z 897.141,A -85,B 0,C 180,E1 5056.807,E2 5056.807} C_VEL
LIN {X 0,Y 426.116,Z 869.548,A -85,B 0,C 180,E1 5056.154,E2 5056.154} C_VEL
LIN {X 0,Y 430.599,Z 846.314,A -85,B 0,C 180,E1 5055.728,E2 5055.728} C_VEL
LIN {X 0,Y 433.744,Z 824.015,A -85,B 0,C 180,E1 5055.375,E2 5055.375} C_VEL
LIN {X 0,Y 439.841,Z 763.942,A -85,B 0,C 180,E1 5054.516,E2 5054.516} C_VEL
LIN {X 0,Y 440.382,Z 756.402,A -85,B 0,C 180,E1 5054.285,E2 5054.285} C_VEL
LIN {X 0,Y 441.061,Z 736.831,A -85,B 0,C 180,E1 5053.212,E2 5053.212} C_VEL
LIN {X 0,Y 441.571,Z 730.35,A -85,B 0,C 180,E1 5053.023,E2 5053.023} C_VEL
LIN {X 0,Y 453.187,Z 618.745,A -85,B 0,C 180,E1 5051.454,E2 5051.454} C_VEL
LIN {X 0,Y 451.058,Z 613.324,A -85,B 0,C 180,E1 5048.991,E2 5048.991} C_VEL
LIN {X 0,Y 449.648,Z 609.556,A -85,B 0,C 180,E1 5046.64,E2 5046.64} C_VEL
LIN {X 0,Y 448.672,Z 606.339,A -85,B 0,C 180,E1 5043.267,E2 5043.267} C_VEL
LIN {X 0,Y 448.949,Z 606.288,A -85,B 0,C 180,E1 5039.684,E2 5039.684} C_VEL
LIN {X 0,Y 449.602,Z 607.134,A -85,B 0,C 180,E1 5037.961,E2 5037.961} C_VEL
LIN {X 0,Y 451.62,Z 611.151,A -85,B 0,C 180,E1 5034.728,E2 5034.728} C_VEL
LIN {X 0,Y 453.529,Z 615.082,A -85,B 0,C 180,E1 5032.653,E2 5032.653} C_VEL
LIN {X 0,Y 454.185,Z 616.665,A -85,B 0,C 180,E1 5032.021,E2 5032.021} C_VEL
LIN {X 0,Y 432.261,Z 824.879,A -85,B 0,C 180,E1 5029.012,E2 5029.012} C_VEL
LIN {X 0,Y 428.928,Z 847.249,A -85,B 0,C 180,E1 5028.65,E2 5028.65} C_VEL
LIN {X 0,Y 423.477,Z 874.064,A -85,B 0,C 180,E1 5028.145,E2 5028.145} C_VEL
LIN {X 0,Y 416.787,Z 899.064,A -85,B 0,C 180,E1 5027.525,E2 5027.525} C_VEL
LIN {X 0,Y 410.342,Z 919.441,A -85,B 0,C 180,E1 5026.902,E2 5026.902} C_VEL
LIN {X 0,Y 402.688,Z 940.444,A -85,B 0,C 180,E1 5026.132,E2 5026.132} C_VEL
LIN {X 0,Y 392.289,Z 965.318,A -85,B 0,C 180,E1 5025.016,E2 5025.016} C_VEL
LIN {X 0,Y 381.607,Z 987.401,A -85,B 0,C 180,E1 5023.798,E2 5023.798} C_VEL
LIN {X 0,Y 371.536,Z 1006.235,A -85,B 0,C 180,E1 5022.558,E2 5022.558} C_VEL
LIN {X 0,Y 360.951,Z 1024.341,A -85,B 0,C 180,E1 5021.152,E2 5021.152} C_VEL
LIN {X 0,Y 346.796,Z 1046.411,A -85,B 0,C 180,E1 5019.09,E2 5019.09} C_VEL
LIN {X 0,Y 333.969,Z 1064.534,A -85,B 0,C 180,E1 5017.017,E2 5017.017} C_VEL
LIN {X 0,Y 322.345,Z 1079.902,A -85,B 0,C 180,E1 5014.924,E2 5014.924} C_VEL
LIN {X 0,Y 310.122,Z 1095.144,A -85,B 0,C 180,E1 5012.453,E2 5012.453} C_VEL
LIN {X 0,Y 295.203,Z 1112.711,A -85,B 0,C 180,E1 5008.973,E2 5008.973} C_VEL
LIN {X 0,Y 282.019,Z 1127.323,A -85,B 0,C 180,E1 5005.339,E2 5005.339} C_VEL
LIN {X 0,Y 271.068,Z 1139.108,A -85,B 0,C 180,E1 5001.783,E2 5001.783} C_VEL
LIN {X 0,Y 259.204,Z 1151.741,A -85,B 0,C 180,E1 4997.131,E2 4997.131} C_VEL
LIN {X 0,Y 248.176,Z 1163.365,A -85,B 0,C 180,E1 4991.664,E2 4991.664} C_VEL
LIN {X 0,Y 240.53,Z 1171.719,A -85,B 0,C 180,E1 4986.769,E2 4986.769} C_VEL
LIN {X 0,Y 234.425,Z 1178.848,A -85,B 0,C 180,E1 4981.642,E2 4981.642} C_VEL
LIN {X 0,Y 229.148,Z 1185.865,A -85,B 0,C 180,E1 4975.316,E2 4975.316} C_VEL
LIN {X 0,Y 225.798,Z 1191.295,A -85,B 0,C 180,E1 4968.592,E2 4968.592} C_VEL
LIN {X 0,Y 224.463,Z 1194.486,A -85,B 0,C 180,E1 4963.131,E2 4963.131} C_VEL
LIN {X 0,Y 224.051,Z 1196.445,A -85,B 0,C 180,E1 4958.21,E2 4958.21} C_VEL
LIN {X 0,Y 223.998,Z 1197.485,A -85,B 0,C 180,E1 4953.582,E2 4953.582} C_VEL
LIN {X 0,Y 224.013,Z 1197.702,A -85,B 0,C 180,E1 4948.721,E2 4948.721} C_VEL
LIN {X 0,Y 224.004,Z 1197.017,A -85,B 0,C 180,E1 4943.85,E2 4943.85} C_VEL
LIN {X 0,Y 224.242,Z 1195.315,A -85,B 0,C 180,E1 4938.685,E2 4938.685} C_VEL
LIN {X 0,Y 225.242,Z 1192.456,A -85,B 0,C 180,E1 4933.229,E2 4933.229} C_VEL
LIN {X 0,Y 227.335,Z 1188.502,A -85,B 0,C 180,E1 4927.774,E2 4927.774} C_VEL
LIN {X 0,Y 230.603,Z 1183.699,A -85,B 0,C 180,E1 4922.638,E2 4922.638} C_VEL
LIN {X 0,Y 235.467,Z 1177.536,A -85,B 0,C 180,E1 4917.364,E2 4917.364} C_VEL
LIN {X 0,Y 243.264,Z 1168.724,A -85,B 0,C 180,E1 4911.335,E2 4911.335} C_VEL
LIN {X 0,Y 253.349,Z 1157.774,A -85,B 0,C 180,E1 4905.59,E2 4905.59} C_VEL
LIN {X 0,Y 262.636,Z 1147.946,A -85,B 0,C 180,E1 4901.409,E2 4901.409} C_VEL
LIN {X 0,Y 273.499,Z 1136.421,A -85,B 0,C 180,E1 4897.365,E2 4897.365} C_VEL
LIN {X 0,Y 288.154,Z 1120.482,A -85,B 0,C 180,E1 4892.888,E2 4892.888} C_VEL
LIN {X 0,Y 300.498,Z 1106.394,A -85,B 0,C 180,E1 4889.72,E2 4889.72} C_VEL
LIN {X 0,Y 312.231,Z 1092.393,A -85,B 0,C 180,E1 4887.094,E2 4887.094} C_VEL
LIN {X 0,Y 325.294,Z 1075.943,A -85,B 0,C 180,E1 4884.517,E2 4884.517} C_VEL
LIN {X 0,Y 340.5,Z 1055.218,A -85,B 0,C 180,E1 4881.885,E2 4881.885} C_VEL
LIN {X 0,Y 352.852,Z 1036.868,A -85,B 0,C 180,E1 4879.979,E2 4879.979} C_VEL
LIN {X 0,Y 364.496,Z 1018.137,A -85,B 0,C 180,E1 4878.351,E2 4878.351} C_VEL
LIN {X 0,Y 377.807,Z 994.445,A -85,B 0,C 180,E1 4876.655,E2 4876.655} C_VEL
LIN {X 0,Y 387.977,Z 974.039,A -85,B 0,C 180,E1 4875.451,E2 4875.451} C_VEL
LIN {X 0,Y 396.584,Z 954.882,A -85,B 0,C 180,E1 4874.499,E2 4874.499} C_VEL
LIN {X 0,Y 404.862,Z 934.221,A -85,B 0,C 180,E1 4873.634,E2 4873.634} C_VEL
LIN {X 0,Y 413.894,Z 908.096,A -85,B 0,C 180,E1 4872.742,E2 4872.742} C_VEL
LIN {X 0,Y 420.702,Z 884.058,A -85,B 0,C 180,E1 4872.095,E2 4872.095} C_VEL
LIN {X 0,Y 425.74,Z 862.577,A -85,B 0,C 180,E1 4871.632,E2 4871.632} C_VEL
LIN {X 0,Y 430.355,Z 837.539,A -85,B 0,C 180,E1 4871.194,E2 4871.194} C_VEL
LIN {X 0,Y 434.745,Z 800.431,A -85,B 0,C 180,E1 4870.631,E2 4870.631} C_VEL
LIN {X 0,Y 453.998,Z 616.263,A -85,B 0,C 180,E1 4867.976,E2 4867.976} C_VEL
LIN {X 0,Y 451.987,Z 612.166,A -85,B 0,C 180,E1 4865.968,E2 4865.968} C_VEL
LIN {X 0,Y 450.666,Z 609.606,A -85,B 0,C 180,E1 4864.326,E2 4864.326} C_VEL
LIN {X 0,Y 449.138,Z 606.509,A -85,B 0,C 180,E1 4861.531,E2 4861.531} C_VEL
LIN {X 0,Y 448.328,Z 605.869,A -85,B 0,C 180,E1 4858.083,E2 4858.083} C_VEL
LIN {X 0,Y 448.523,Z 606.528,A -85,B 0,C 180,E1 4855.909,E2 4855.909} C_VEL
LIN {X 0,Y 449.847,Z 610.496,A -85,B 0,C 180,E1 4852.4,E2 4852.4} C_VEL
LIN {X 0,Y 451.821,Z 615.62,A -85,B 0,C 180,E1 4849.674,E2 4849.674} C_VEL
LIN {X 0,Y 452.987,Z 618.766,A -85,B 0,C 180,E1 4848.426,E2 4848.426} C_VEL
LIN {X 0,Y 431.11,Z 828.848,A -85,B 0,C 180,E1 4845.492,E2 4845.492} C_VEL
LIN {X 0,Y 426.885,Z 855.775,A -85,B 0,C 180,E1 4845.059,E2 4845.059} C_VEL
LIN {X 0,Y 421.145,Z 881.291,A -85,B 0,C 180,E1 4844.547,E2 4844.547} C_VEL
LIN {X 0,Y 415.701,Z 901.119,A -85,B 0,C 180,E1 4844.053,E2 4844.053} C_VEL
LIN {X 0,Y 408.67,Z 922.922,A -85,B 0,C 180,E1 4843.383,E2 4843.383} C_VEL
LIN {X 0,Y 398.674,Z 949.103,A -85,B 0,C 180,E1 4842.373,E2 4842.373} C_VEL
LIN {X 0,Y 389.781,Z 969.179,A -85,B 0,C 180,E1 4841.416,E2 4841.416} C_VEL
LIN {X 0,Y 380.534,Z 987.867,A -85,B 0,C 180,E1 4840.365,E2 4840.365} C_VEL
LIN {X 0,Y 369.069,Z 1008.8,A -85,B 0,C 180,E1 4838.959,E2 4838.959} C_VEL
LIN {X 0,Y 355.415,Z 1030.907,A -85,B 0,C 180,E1 4837.124,E2 4837.124} C_VEL
LIN {X 0,Y 343.694,Z 1048.176,A -85,B 0,C 180,E1 4835.386,E2 4835.386} C_VEL
LIN {X 0,Y 331.516,Z 1064.788,A -85,B 0,C 180,E1 4833.386,E2 4833.386} C_VEL
LIN {X 0,Y 315.943,Z 1084.265,A -85,B 0,C 180,E1 4830.495,E2 4830.495} C_VEL
LIN {X 0,Y 303.521,Z 1098.658,A -85,B 0,C 180,E1 4827.847,E2 4827.847} C_VEL
LIN {X 0,Y 291.78,Z 1111.553,A -85,B 0,C 180,E1 4824.986,E2 4824.986} C_VEL
LIN {X 0,Y 277.873,Z 1126.113,A -85,B 0,C 180,E1 4821.009,E2 4821.009} C_VEL
LIN {X 0,Y 265.544,Z 1138.329,A -85,B 0,C 180,E1 4816.74,E2 4816.74} C_VEL
LIN {X 0,Y 255.682,Z 1147.958,A -85,B 0,C 180,E1 4812.574,E2 4812.574} C_VEL
LIN {X 0,Y 245.385,Z 1158.083,A -85,B 0,C 180,E1 4807.09,E2 4807.09} C_VEL
LIN {X 0,Y 237.154,Z 1166.234,A -85,B 0,C 180,E1 4801.238,E2 4801.238} C_VEL
LIN {X 0,Y 231.707,Z 1172.105,A -85,B 0,C 180,E1 4795.839,E2 4795.839} C_VEL
LIN {X 0,Y 227.351,Z 1177.541,A -85,B 0,C 180,E1 4789.26,E2 4789.26} C_VEL
LIN {X 0,Y 225.057,Z 1181.039,A -85,B 0,C 180,E1 4782.835,E2 4782.835} C_VEL
LIN {X 0,Y 224.284,Z 1182.85,A -85,B 0,C 180,E1 4777.686,E2 4777.686} C_VEL
LIN {X 0,Y 224.058,Z 1183.733,A -85,B 0,C 180,E1 4772.814,E2 4772.814} C_VEL
LIN {X 0,Y 224.05,Z 1183.829,A -85,B 0,C 180,E1 4768.21,E2 4768.21} C_VEL
LIN {X 0,Y 224.197,Z 1183.14,A -85,B 0,C 180,E1 4763.342,E2 4763.342} C_VEL
LIN {X 0,Y 224.776,Z 1181.633,A -85,B 0,C 180,E1 4758.453,E2 4758.453} C_VEL
LIN {X 0,Y 226.299,Z 1178.985,A -85,B 0,C 180,E1 4753.046,E2 4753.046} C_VEL
LIN {X 0,Y 229.034,Z 1175.292,A -85,B 0,C 180,E1 4747.679,E2 4747.679} C_VEL
LIN {X 0,Y 234.149,Z 1169.544,A -85,B 0,C 180,E1 4741.428,E2 4741.428} C_VEL
LIN {X 0,Y 241.721,Z 1161.668,A -85,B 0,C 180,E1 4735.192,E2 4735.192} C_VEL
LIN {X 0,Y 249.542,Z 1153.997,A -85,B 0,C 180,E1 4730.426,E2 4730.426} C_VEL
LIN {X 0,Y 259.751,Z 1144.156,A -85,B 0,C 180,E1 4725.527,E2 4725.527} C_VEL
LIN {X 0,Y 272.103,Z 1131.968,A -85,B 0,C 180,E1 4720.803,E2 4720.803} C_VEL
LIN {X 0,Y 283.609,Z 1120.273,A -85,B 0,C 180,E1 4717.178,E2 4717.178} C_VEL
LIN {X 0,Y 295.466,Z 1107.754,A -85,B 0,C 180,E1 4713.995,E2 4713.995} C_VEL
LIN {X 0,Y 310.881,Z 1090.454,A -85,B 0,C 180,E1 4710.463,E2 4710.463} C_VEL
LIN {X 0,Y 323.679,Z 1074.98,A -85,B 0,C 180,E1 4707.935,E2 4707.935} C_VEL
LIN {X 0,Y 335.92,Z 1059.169,A -85,B 0,C 180,E1 4705.79,E2 4705.79} C_VEL
LIN {X 0,Y 350.176,Z 1039.213,A -85,B 0,C 180,E1 4703.563,E2 4703.563} C_VEL
LIN {X 0,Y 362.451,Z 1020.109,A -85,B 0,C 180,E1 4701.832,E2 4701.832} C_VEL
LIN {X 0,Y 372.587,Z 1002.904,A -85,B 0,C 180,E1 4700.516,E2 4700.516} C_VEL
LIN {X 0,Y 382.922,Z 983.664,A -85,B 0,C 180,E1 4699.277,E2 4699.277} C_VEL
LIN {X 0,Y 394.904,Z 958.415,A -85,B 0,C 180,E1 4697.947,E2 4697.947} C_VEL
LIN {X 0,Y 403.672,Z 937.089,A -85,B 0,C 180,E1 4697.041,E2 4697.041} C_VEL
LIN {X 0,Y 410.566,Z 917.994,A -85,B 0,C 180,E1 4696.357,E2 4696.357} C_VEL
LIN {X 0,Y 417.743,Z 894.993,A -85,B 0,C 180,E1 4695.68,E2 4695.68} C_VEL
LIN {X 0,Y 424.573,Z 867.717,A -85,B 0,C 180,E1 4695.066,E2 4695.066} C_VEL
LIN {X 0,Y 428.871,Z 845.498,A -85,B 0,C 180,E1 4694.673,E2 4694.673} C_VEL
LIN {X 0,Y 432.109,Z 822.592,A -85,B 0,C 180,E1 4694.319,E2 4694.319} C_VEL
LIN {X 0,Y 441.571,Z 730.35,A -85,B 0,C 180,E1 4693.023,E2 4693.023} C_VEL
LIN {X 0,Y 442.157,Z 722.819,A -85,B 0,C 180,E1 4692.788,E2 4692.788} C_VEL
LIN {X 0,Y 443.094,Z 703.258,A -85,B 0,C 180,E1 4691.721,E2 4691.721} C_VEL
LIN {X 0,Y 443.654,Z 696.778,A -85,B 0,C 180,E1 4691.537,E2 4691.537} C_VEL
LIN {X 0,Y 451.294,Z 624.796,A -85,B 0,C 180,E1 4690.532,E2 4690.532} C_VEL
LIN {X 0,Y 449.279,Z 619.333,A -85,B 0,C 180,E1 4687.803,E2 4687.803} C_VEL
LIN {X 0,Y 448.49,Z 617.195,A -85,B 0,C 180,E1 4686.272,E2 4686.272} C_VEL
LIN {X 0,Y 447.682,Z 614.267,A -85,B 0,C 180,E1 4683.201,E2 4683.201} C_VEL
LIN {X 0,Y 447.987,Z 614.249,A -85,B 0,C 180,E1 4679.616,E2 4679.616} C_VEL
LIN {X 0,Y 448.559,Z 615.011,A -85,B 0,C 180,E1 4678.084,E2 4678.084} C_VEL
LIN {X 0,Y 450.514,Z 619.06,A -85,B 0,C 180,E1 4674.843,E2 4674.843} C_VEL
LIN {X 0,Y 452.209,Z 622.647,A -85,B 0,C 180,E1 4672.939,E2 4672.939} C_VEL
LIN {X 0,Y 430.337,Z 826.582,A -85,B 0,C 180,E1 4670.028,E2 4670.028} C_VEL
LIN {X 0,Y 426.55,Z 850.894,A -85,B 0,C 180,E1 4669.638,E2 4669.638} C_VEL
LIN {X 0,Y 420.394,Z 878.918,A -85,B 0,C 180,E1 4669.1,E2 4669.1} C_VEL
LIN {X 0,Y 414.428,Z 900.572,A -85,B 0,C 180,E1 4668.562,E2 4668.562} C_VEL
LIN {X 0,Y 407.926,Z 920.669,A -85,B 0,C 180,E1 4667.957,E2 4667.957} C_VEL
LIN {X 0,Y 399.657,Z 942.849,A -85,B 0,C 180,E1 4667.153,E2 4667.153} C_VEL
LIN {X 0,Y 388.494,Z 968.503,A -85,B 0,C 180,E1 4665.998,E2 4665.998} C_VEL
LIN {X 0,Y 378.516,Z 988.645,A -85,B 0,C 180,E1 4664.895,E2 4664.895} C_VEL
LIN {X 0,Y 368.295,Z 1007.33,A -85,B 0,C 180,E1 4663.679,E2 4663.679} C_VEL
LIN {X 0,Y 355.346,Z 1028.906,A -85,B 0,C 180,E1 4662.001,E2 4662.001} C_VEL
LIN {X 0,Y 341.492,Z 1049.464,A -85,B 0,C 180,E1 4660.03,E2 4660.03} C_VEL
LIN {X 0,Y 329.621,Z 1065.76,A -85,B 0,C 180,E1 4658.158,E2 4658.158} C_VEL
LIN {X 0,Y 317.001,Z 1081.953,A -85,B 0,C 180,E1 4655.941,E2 4655.941} C_VEL
LIN {X 0,Y 301.325,Z 1100.73,A -85,B 0,C 180,E1 4652.784,E2 4652.784} C_VEL
LIN {X 0,Y 287.599,Z 1116.013,A -85,B 0,C 180,E1 4649.564,E2 4649.564} C_VEL
LIN {X 0,Y 275.621,Z 1128.804,A -85,B 0,C 180,E1 4646.286,E2 4646.286} C_VEL
LIN {X 0,Y 261.99,Z 1142.958,A -85,B 0,C 180,E1 4641.83,E2 4641.83} C_VEL
LIN {X 0,Y 249.339,Z 1155.584,A -85,B 0,C 180,E1 4636.706,E2 4636.706} C_VEL
LIN {X 0,Y 240.275,Z 1164.778,A -85,B 0,C 180,E1 4632.065,E2 4632.065} C_VEL
LIN {X 0,Y 231.817,Z 1173.658,A -85,B 0,C 180,E1 4626.528,E2 4626.528} C_VEL
LIN {X 0,Y 224.307,Z 1182.17,A -85,B 0,C 180,E1 4619.628,E2 4619.628} C_VEL
LIN {X 0,Y 220.149,Z 1187.622,A -85,B 0,C 180,E1 4613.842,E2 4613.842} C_VEL
LIN {X 0,Y 217.731,Z 1191.549,A -85,B 0,C 180,E1 4608.473,E2 4608.473} C_VEL
LIN {X 0,Y 216.491,Z 1194.355,A -85,B 0,C 180,E1 4603.351,E2 4603.351} C_VEL
LIN {X 0,Y 216.054,Z 1196.269,A -85,B 0,C 180,E1 4598.248,E2 4598.248} C_VEL
LIN {X 0,Y 216.003,Z 1197.263,A -85,B 0,C 180,E1 4593.449,E2 4593.449} C_VEL
LIN {X 0,Y 216.016,Z 1197.455,A -85,B 0,C 180,E1 4588.673,E2 4588.673} C_VEL
LIN {X 0,Y 216.009,Z 1196.768,A -85,B 0,C 180,E1 4583.621,E2 4583.621} C_VEL
LIN {X 0,Y 216.279,Z 1195.064,A -85,B 0,C 180,E1 4578.263,E2 4578.263} C_VEL
LIN {X 0,Y 217.397,Z 1192.201,A -85,B 0,C 180,E1 4572.605,E2 4572.605} C_VEL
LIN {X 0,Y 219.698,Z 1188.244,A -85,B 0,C 180,E1 4566.958,E2 4566.958} C_VEL
LIN {X 0,Y 223.223,Z 1183.438,A -85,B 0,C 180,E1 4561.653,E2 4561.653} C_VEL
LIN {X 0,Y 228.445,Z 1177.273,A -85,B 0,C 180,E1 4556.229,E2 4556.229} C_VEL
LIN {X 0,Y 236.734,Z 1168.458,A -85,B 0,C 180,E1 4550.059,E2 4550.059} C_VEL
LIN {X 0,Y 247.231,Z 1157.647,A -85,B 0,C 180,E1 4544.287,E2 4544.287} C_VEL
LIN {X 0,Y 257.11,Z 1147.67,A -85,B 0,C 180,E1 4539.993,E2 4539.993} C_VEL
LIN {X 0,Y 268.213,Z 1136.376,A -85,B 0,C 180,E1 4536.005,E2 4536.005} C_VEL
LIN {X 0,Y 283.012,Z 1120.908,A -85,B 0,C 180,E1 4531.629,E2 4531.629} C_VEL
LIN {X 0,Y 296.412,Z 1106.097,A -85,B 0,C 180,E1 4528.306,E2 4528.306} C_VEL
LIN {X 0,Y 308.495,Z 1092.087,A -85,B 0,C 180,E1 4525.704,E2 4525.704} C_VEL
LIN {X 0,Y 322.163,Z 1075.314,A -85,B 0,C 180,E1 4523.115,E2 4523.115} C_VEL
LIN {X 0,Y 337.479,Z 1054.876,A -85,B 0,C 180,E1 4520.57,E2 4520.57} C_VEL
LIN {X 0,Y 349.561,Z 1037.319,A -85,B 0,C 180,E1 4518.775,E2 4518.775} C_VEL
LIN {X 0,Y 361.133,Z 1019.114,A -85,B 0,C 180,E1 4517.212,E2 4517.212} C_VEL
LIN {X 0,Y 374.196,Z 996.57,A -85,B 0,C 180,E1 4515.607,E2 4515.607} C_VEL
LIN {X 0,Y 385.432,Z 974.477,A -85,B 0,C 180,E1 4514.32,E2 4514.32} C_VEL
LIN {X 0,Y 394.171,Z 955.38,A -85,B 0,C 180,E1 4513.391,E2 4513.391} C_VEL
LIN {X 0,Y 402.306,Z 935.459,A -85,B 0,C 180,E1 4512.572,E2 4512.572} C_VEL
LIN {X 0,Y 411.052,Z 910.981,A -85,B 0,C 180,E1 4511.741,E2 4511.741} C_VEL
LIN {X 0,Y 418.587,Z 885.06,A -85,B 0,C 180,E1 4511.05,E2 4511.05} C_VEL
LIN {X 0,Y 423.775,Z 863.36,A -85,B 0,C 180,E1 4510.592,E2 4510.592} C_VEL
LIN {X 0,Y 428.201,Z 839.953,A -85,B 0,C 180,E1 4510.188,E2 4510.188} C_VEL
LIN {X 0,Y 432.638,Z 804.58,A -85,B 0,C 180,E1 4509.654,E2 4509.654} C_VEL
LIN {X 0,Y 451.996,Z 622.435,A -85,B 0,C 180,E1 4507.052,E2 4507.052} C_VEL
LIN {X 0,Y 449.87,Z 617.913,A -85,B 0,C 180,E1 4504.589,E2 4504.589} C_VEL
LIN {X 0,Y 448.162,Z 614.458,A -85,B 0,C 180,E1 4501.534,E2 4501.534} C_VEL
LIN {X 0,Y 447.353,Z 613.811,A -85,B 0,C 180,E1 4498.079,E2 4498.079} C_VEL
LIN {X 0,Y 447.523,Z 614.412,A -85,B 0,C 180,E1 4496.028,E2 4496.028} C_VEL
LIN {X 0,Y 448.754,Z 618.306,A -85,B 0,C 180,E1 4492.575,E2 4492.575} C_VEL
LIN {X 0,Y 450.666,Z 623.448,A -85,B 0,C 180,E1 4489.841,E2 4489.841} C_VEL
LIN {X 0,Y 451.065,Z 624.881,A -85,B 0,C 180,E1 4489.347,E2 4489.347} C_VEL
LIN {X 0,Y 429.386,Z 829.144,A -85,B 0,C 180,E1 4486.532,E2 4486.532} C_VEL
LIN {X 0,Y 425.028,Z 856.265,A -85,B 0,C 180,E1 4486.104,E2 4486.104} C_VEL
LIN {X 0,Y 419.307,Z 881.339,A -85,B 0,C 180,E1 4485.613,E2 4485.613} C_VEL
LIN {X 0,Y 413.582,Z 901.853,A -85,B 0,C 180,E1 4485.114,E2 4485.114} C_VEL
LIN {X 0,Y 405.892,Z 925.209,A -85,B 0,C 180,E1 4484.407,E2 4484.407} C_VEL
LIN {X 0,Y 395.843,Z 950.702,A -85,B 0,C 180,E1 4483.43,E2 4483.43} C_VEL
LIN {X 0,Y 386.867,Z 970.527,A -85,B 0,C 180,E1 4482.497,E2 4482.497} C_VEL
LIN {X 0,Y 377.455,Z 989.139,A -85,B 0,C 180,E1 4481.465,E2 4481.465} C_VEL
LIN {X 0,Y 364.882,Z 1011.524,A -85,B 0,C 180,E1 4479.968,E2 4479.968} C_VEL
LIN {X 0,Y 351.935,Z 1031.856,A -85,B 0,C 180,E1 4478.285,E2 4478.285} C_VEL
LIN {X 0,Y 340.457,Z 1048.408,A -85,B 0,C 180,E1 4476.641,E2 4476.641} C_VEL
LIN {X 0,Y 327.999,Z 1065.029,A -85,B 0,C 180,E1 4474.67,E2 4474.67} C_VEL
LIN {X 0,Y 311.989,Z 1084.558,A -85,B 0,C 180,E1 4471.804,E2 4471.804} C_VEL
LIN {X 0,Y 299.231,Z 1098.946,A -85,B 0,C 180,E1 4469.179,E2 4469.179} C_VEL
LIN {X 0,Y 287.134,Z 1111.835,A -85,B 0,C 180,E1 4466.332,E2 4466.332} C_VEL
LIN {X 0,Y 272.753,Z 1126.382,A -85,B 0,C 180,E1 4462.357,E2 4462.357} C_VEL
LIN {X 0,Y 260.265,Z 1138.297,A -85,B 0,C 180,E1 4458.186,E2 4458.186} C_VEL
LIN {X 0,Y 250.132,Z 1147.778,A -85,B 0,C 180,E1 4454.072,E2 4454.072} C_VEL
LIN {X 0,Y 239.5,Z 1157.726,A -85,B 0,C 180,E1 4448.674,E2 4448.674} C_VEL
LIN {X 0,Y 230.449,Z 1166.199,A -85,B 0,C 180,E1 4442.549,E2 4442.549} C_VEL
LIN {X 0,Y 224.645,Z 1172.031,A -85,B 0,C 180,E1 4437.101,E2 4437.101} C_VEL
LIN {X 0,Y 220.232,Z 1177.025,A -85,B 0,C 180,E1 4431.019,E2 4431.019} C_VEL
LIN {X 0,Y 217.299,Z 1181.076,A -85,B 0,C 180,E1 4423.844,E2 4423.844} C_VEL
LIN {X 0,Y 216.339,Z 1183.035,A -85,B 0,C 180,E1 4418.238,E2 4418.238} C_VEL
LIN {X 0,Y 216.066,Z 1183.959,A -85,B 0,C 180,E1 4413.184,E2 4413.184} C_VEL
LIN {X 0,Y 216.053,Z 1184.097,A -85,B 0,C 180,E1 4408.409,E2 4408.409} C_VEL
LIN {X 0,Y 216.2,Z 1183.452,A -85,B 0,C 180,E1 4403.361,E2 4403.361} C_VEL
LIN {X 0,Y 216.853,Z 1181.883,A -85,B 0,C 180,E1 4398.025,E2 4398.025} C_VEL
LIN {X 0,Y 218.519,Z 1179.236,A -85,B 0,C 180,E1 4392.423,E2 4392.423} C_VEL
LIN {X 0,Y 221.476,Z 1175.545,A -85,B 0,C 180,E1 4386.874,E2 4386.874} C_VEL
LIN {X 0,Y 226.95,Z 1169.798,A -85,B 0,C 180,E1 4380.434,E2 4380.434} C_VEL
LIN {X 0,Y 234.985,Z 1161.927,A -85,B 0,C 180,E1 4374.042,E2 4374.042} C_VEL
LIN {X 0,Y 243.358,Z 1154.131,A -85,B 0,C 180,E1 4369.114,E2 4369.114} C_VEL
LIN {X 0,Y 254.416,Z 1143.971,A -85,B 0,C 180,E1 4364.012,E2 4364.012} C_VEL
LIN {X 0,Y 267.346,Z 1131.677,A -85,B 0,C 180,E1 4359.27,E2 4359.27} C_VEL
LIN {X 0,Y 278.979,Z 1120.265,A -85,B 0,C 180,E1 4355.747,E2 4355.747} C_VEL
LIN {X 0,Y 291.606,Z 1107.342,A -85,B 0,C 180,E1 4352.489,E2 4352.489} C_VEL
LIN {X 0,Y 307.68,Z 1089.715,A -85,B 0,C 180,E1 4348.961,E2 4348.961} C_VEL
LIN {X 0,Y 320.667,Z 1074.369,A -85,B 0,C 180,E1 4346.505,E2 4346.505} C_VEL
LIN {X 0,Y 333.608,Z 1057.979,A -85,B 0,C 180,E1 4344.338,E2 4344.338} C_VEL
LIN {X 0,Y 349.002,Z 1036.54,A -85,B 0,C 180,E1 4342.044,E2 4342.044} C_VEL
LIN {X 0,Y 360.334,Z 1019.148,A -85,B 0,C 180,E1 4340.527,E2 4340.527} C_VEL
LIN {X 0,Y 370.671,Z 1001.832,A -85,B 0,C 180,E1 4339.246,E2 4339.246} C_VEL
LIN {X 0,Y 382.466,Z 980.06,A -85,B 0,C 180,E1 4337.9,E2 4337.9} C_VEL
LIN {X 0,Y 393.588,Z 956.397,A -85,B 0,C 180,E1 4336.719,E2 4336.719} C_VEL
LIN {X 0,Y 401.835,Z 936.515,A -85,B 0,C 180,E1 4335.905,E2 4335.905} C_VEL
LIN {X 0,Y 408.831,Z 917.338,A -85,B 0,C 180,E1 4335.243,E2 4335.243} C_VEL
LIN {X 0,Y 416.551,Z 892.772,A -85,B 0,C 180,E1 4334.547,E2 4334.547} C_VEL
LIN {X 0,Y 423.048,Z 866.531,A -85,B 0,C 180,E1 4333.984,E2 4333.984} C_VEL
LIN {X 0,Y 427.289,Z 844.692,A -85,B 0,C 180,E1 4333.611,E2 4333.611} C_VEL
LIN {X 0,Y 430.728,Z 820.327,A -85,B 0,C 180,E1 4333.243,E2 4333.243} C_VEL
LIN {X 0,Y 443.654,Z 696.778,A -85,B 0,C 180,E1 4331.537,E2 4331.537} C_VEL
LIN {X 0,Y 444.291,Z 689.246,A -85,B 0,C 180,E1 4331.308,E2 4331.308} C_VEL
LIN {X 0,Y 445.433,Z 669.698,A -85,B 0,C 180,E1 4330.245,E2 4330.245} C_VEL
LIN {X 0,Y 446.025,Z 663.222,A -85,B 0,C 180,E1 4330.06,E2 4330.06} C_VEL
LIN {X 0,Y 449.514,Z 630.887,A -85,B 0,C 180,E1 4329.604,E2 4329.604} C_VEL
LIN {X 0,Y 447.885,Z 626.192,A -85,B 0,C 180,E1 4327.053,E2 4327.053} C_VEL
LIN {X 0,Y 446.708,Z 622.213,A -85,B 0,C 180,E1 4323.208,E2 4323.208} C_VEL
LIN {X 0,Y 446.968,Z 622.158,A -85,B 0,C 180,E1 4319.744,E2 4319.744} C_VEL
LIN {X 0,Y 447.518,Z 622.888,A -85,B 0,C 180,E1 4318.207,E2 4318.207} C_VEL
LIN {X 0,Y 449.363,Z 626.855,A -85,B 0,C 180,E1 4315.022,E2 4315.022} C_VEL
LIN {X 0,Y 450.306,Z 629.044,A -85,B 0,C 180,E1 4313.858,E2 4313.858} C_VEL
LIN {X 0,Y 428.634,Z 827.632,A -85,B 0,C 180,E1 4311.063,E2 4311.063} C_VEL
LIN {X 0,Y 424.297,Z 854.5,A -85,B 0,C 180,E1 4310.638,E2 4310.638} C_VEL
LIN {X 0,Y 418.256,Z 880.643,A -85,B 0,C 180,E1 4310.135,E2 4310.135} C_VEL
LIN {X 0,Y 412.433,Z 901.338,A -85,B 0,C 180,E1 4309.631,E2 4309.631} C_VEL
LIN {X 0,Y 405.396,Z 922.631,A -85,B 0,C 180,E1 4309,E2 4309} C_VEL
LIN {X 0,Y 395.496,Z 948.216,A -85,B 0,C 180,E1 4308.067,E2 4308.067} C_VEL
LIN {X 0,Y 385.259,Z 970.779,A -85,B 0,C 180,E1 4307.044,E2 4307.044} C_VEL
LIN {X 0,Y 375.547,Z 989.924,A -85,B 0,C 180,E1 4306.007,E2 4306.007} C_VEL
LIN {X 0,Y 363.908,Z 1010.66,A -85,B 0,C 180,E1 4304.666,E2 4304.666} C_VEL
LIN {X 0,Y 349.498,Z 1033.528,A -85,B 0,C 180,E1 4302.849,E2 4302.849} C_VEL
LIN {X 0,Y 337.309,Z 1051.098,A -85,B 0,C 180,E1 4301.149,E2 4301.149} C_VEL
LIN {X 0,Y 325.175,Z 1067.293,A -85,B 0,C 180,E1 4299.291,E2 4299.291} C_VEL
LIN {X 0,Y 310.242,Z 1085.89,A -85,B 0,C 180,E1 4296.71,E2 4296.71} C_VEL
LIN {X 0,Y 295.388,Z 1102.803,A -85,B 0,C 180,E1 4293.767,E2 4293.767} C_VEL
LIN {X 0,Y 282.728,Z 1116.446,A -85,B 0,C 180,E1 4290.87,E2 4290.87} C_VEL
LIN {X 0,Y 270.189,Z 1129.366,A -85,B 0,C 180,E1 4287.537,E2 4287.537} C_VEL
LIN {X 0,Y 255.697,Z 1143.768,A -85,B 0,C 180,E1 4282.912,E2 4282.912} C_VEL
LIN {X 0,Y 243.363,Z 1155.554,A -85,B 0,C 180,E1 4278.043,E2 4278.043} C_VEL
LIN {X 0,Y 233.998,Z 1164.579,A -85,B 0,C 180,E1 4273.412,E2 4273.412} C_VEL
LIN {X 0,Y 225.462,Z 1173.026,A -85,B 0,C 180,E1 4268.056,E2 4268.056} C_VEL
LIN {X 0,Y 217.109,Z 1181.885,A -85,B 0,C 180,E1 4260.743,E2 4260.743} C_VEL
LIN {X 0,Y 212.586,Z 1187.365,A -85,B 0,C 180,E1 4254.746,E2 4254.746} C_VEL
LIN {X 0,Y 209.842,Z 1191.464,A -85,B 0,C 180,E1 4248.905,E2 4248.905} C_VEL
LIN {X 0,Y 208.521,Z 1194.225,A -85,B 0,C 180,E1 4243.589,E2 4243.589} C_VEL
LIN {X 0,Y 208.065,Z 1196.019,A -85,B 0,C 180,E1 4238.567,E2 4238.567} C_VEL
LIN {X 0,Y 208.005,Z 1197.016,A -85,B 0,C 180,E1 4233.582,E2 4233.582} C_VEL
LIN {X 0,Y 208.02,Z 1197.207,A -85,B 0,C 180,E1 4228.622,E2 4228.622} C_VEL
LIN {X 0,Y 208.014,Z 1196.519,A -85,B 0,C 180,E1 4223.375,E2 4223.375} C_VEL
LIN {X 0,Y 208.326,Z 1194.811,A -85,B 0,C 180,E1 4217.808,E2 4217.808} C_VEL
LIN {X 0,Y 209.572,Z 1191.945,A -85,B 0,C 180,E1 4211.933,E2 4211.933} C_VEL
LIN {X 0,Y 212.104,Z 1187.986,A -85,B 0,C 180,E1 4206.082,E2 4206.082} C_VEL
LIN {X 0,Y 216.143,Z 1182.911,A -85,B 0,C 180,E1 4200.331,E2 4200.331} C_VEL
LIN {X 0,Y 222.139,Z 1176.376,A -85,B 0,C 180,E1 4194.503,E2 4194.503} C_VEL
LIN {X 0,Y 232.378,Z 1166.12,A -85,B 0,C 180,E1 4187.503,E2 4187.503} C_VEL
LIN {X 0,Y 241.88,Z 1156.9,A -85,B 0,C 180,E1 4182.623,E2 4182.623} C_VEL
LIN {X 0,Y 252.305,Z 1146.863,A -85,B 0,C 180,E1 4178.309,E2 4178.309} C_VEL
LIN {X 0,Y 265.801,Z 1133.74,A -85,B 0,C 180,E1 4173.762,E2 4173.762} C_VEL
LIN {X 0,Y 280.69,Z 1118.463,A -85,B 0,C 180,E1 4169.636,E2 4169.636} C_VEL
LIN {X 0,Y 293.225,Z 1105.01,A -85,B 0,C 180,E1 4166.695,E2 4166.695} C_VEL
LIN {X 0,Y 305.733,Z 1090.876,A -85,B 0,C 180,E1 4164.13,E2 4164.13} C_VEL
LIN {X 0,Y 321.21,Z 1072.265,A -85,B 0,C 180,E1 4161.359,E2 4161.359} C_VEL
LIN {X 0,Y 335.455,Z 1053.405,A -85,B 0,C 180,E1 4159.113,E2 4159.113} C_VEL
LIN {X 0,Y 347.396,Z 1036.335,A -85,B 0,C 180,E1 4157.418,E2 4157.418} C_VEL
LIN {X 0,Y 359.618,Z 1017.379,A -85,B 0,C 180,E1 4155.842,E2 4155.842} C_VEL
LIN {X 0,Y 373.839,Z 992.75,A -85,B 0,C 180,E1 4154.175,E2 4154.175} C_VEL
LIN {X 0,Y 383.921,Z 973.093,A -85,B 0,C 180,E1 4153.083,E2 4153.083} C_VEL
LIN {X 0,Y 392.798,Z 953.845,A -85,B 0,C 180,E1 4152.181,E2 4152.181} C_VEL
LIN {X 0,Y 402.143,Z 930.985,A -85,B 0,C 180,E1 4151.288,E2 4151.288} C_VEL
LIN {X 0,Y 411.107,Z 904.944,A -85,B 0,C 180,E1 4150.475,E2 4150.475} C_VEL
LIN {X 0,Y 417.421,Z 882.95,A -85,B 0,C 180,E1 4149.924,E2 4149.924} C_VEL
LIN {X 0,Y 422.63,Z 861.039,A -85,B 0,C 180,E1 4149.484,E2 4149.484} C_VEL
LIN {X 0,Y 427.633,Z 833.584,A -85,B 0,C 180,E1 4149.033,E2 4149.033} C_VEL
LIN {X 0,Y 433.146,Z 785.484,A -85,B 0,C 180,E1 4148.339,E2 4148.339} C_VEL
LIN {X 0,Y 450.107,Z 628.615,A -85,B 0,C 180,E1 4146.121,E2 4146.121} C_VEL
LIN {X 0,Y 448.506,Z 625.353,A -85,B 0,C 180,E1 4144.091,E2 4144.091} C_VEL
LIN {X 0,Y 447.126,Z 622.355,A -85,B 0,C 180,E1 4141.41,E2 4141.41} C_VEL
LIN {X 0,Y 446.375,Z 621.771,A -85,B 0,C 180,E1 4137.946,E2 4137.946} C_VEL
LIN {X 0,Y 446.539,Z 622.441,A -85,B 0,C 180,E1 4136.02,E2 4136.02} C_VEL
LIN {X 0,Y 447.697,Z 626.224,A -85,B 0,C 180,E1 4132.686,E2 4132.686} C_VEL
LIN {X 0,Y 449.282,Z 630.788,A -85,B 0,C 180,E1 4130.278,E2 4130.278} C_VEL
LIN {X 0,Y 427.842,Z 829.148,A -85,B 0,C 180,E1 4127.585,E2 4127.585} C_VEL
LIN {X 0,Y 423.434,Z 856.204,A -85,B 0,C 180,E1 4127.167,E2 4127.167} C_VEL
LIN {X 0,Y 417.619,Z 881.373,A -85,B 0,C 180,E1 4126.688,E2 4126.688} C_VEL
LIN {X 0,Y 411.83,Z 901.851,A -85,B 0,C 180,E1 4126.206,E2 4126.206} C_VEL
LIN {X 0,Y 404.165,Z 924.85,A -85,B 0,C 180,E1 4125.53,E2 4125.53} C_VEL
LIN {X 0,Y 394.117,Z 950.112,A -85,B 0,C 180,E1 4124.594,E2 4124.594} C_VEL
LIN {X 0,Y 384.961,Z 970.095,A -85,B 0,C 180,E1 4123.683,E2 4123.683} C_VEL
LIN {X 0,Y 375.468,Z 988.628,A -85,B 0,C 180,E1 4122.688,E2 4122.688} C_VEL
LIN {X 0,Y 362.913,Z 1010.733,A -85,B 0,C 180,E1 4121.257,E2 4121.257} C_VEL
LIN {X 0,Y 349.283,Z 1031.807,A -85,B 0,C 180,E1 4119.559,E2 4119.559} C_VEL
LIN {X 0,Y 337.644,Z 1048.289,A -85,B 0,C 180,E1 4117.957,E2 4117.957} C_VEL
LIN {X 0,Y 325.021,Z 1064.797,A -85,B 0,C 180,E1 4116.041,E2 4116.041} C_VEL
LIN {X 0,Y 308.744,Z 1084.249,A -85,B 0,C 180,E1 4113.246,E2 4113.246} C_VEL
LIN {X 0,Y 295.819,Z 1098.475,A -85,B 0,C 180,E1 4110.698,E2 4110.698} C_VEL
LIN {X 0,Y 283.326,Z 1111.429,A -85,B 0,C 180,E1 4107.885,E2 4107.885} C_VEL
LIN {X 0,Y 268.414,Z 1126.091,A -85,B 0,C 180,E1 4103.936,E2 4103.936} C_VEL
LIN {X 0,Y 254.827,Z 1138.563,A -85,B 0,C 180,E1 4099.571,E2 4099.571} C_VEL
LIN {X 0,Y 244.256,Z 1148.041,A -85,B 0,C 180,E1 4095.421,E2 4095.421} C_VEL
LIN {X 0,Y 232.822,Z 1158.25,A -85,B 0,C 180,E1 4089.785,E2 4089.785} C_VEL
LIN {X 0,Y 223.542,Z 1166.456,A -85,B 0,C 180,E1 4083.686,E2 4083.686} C_VEL
LIN {X 0,Y 217.516,Z 1172.128,A -85,B 0,C 180,E1 4078.26,E2 4078.26} C_VEL
LIN {X 0,Y 212.916,Z 1176.917,A -85,B 0,C 180,E1 4072.309,E2 4072.309} C_VEL
LIN {X 0,Y 209.595,Z 1181.113,A -85,B 0,C 180,E1 4064.929,E2 4064.929} C_VEL
LIN {X 0,Y 208.396,Z 1183.242,A -85,B 0,C 180,E1 4058.736,E2 4058.736} C_VEL
LIN {X 0,Y 208.072,Z 1184.206,A -85,B 0,C 180,E1 4053.306,E2 4053.306} C_VEL
LIN {X 0,Y 208.057,Z 1184.344,A -85,B 0,C 180,E1 4048.348,E2 4048.348} C_VEL
LIN {X 0,Y 208.222,Z 1183.7,A -85,B 0,C 180,E1 4043.106,E2 4043.106} C_VEL
LIN {X 0,Y 208.964,Z 1182.092,A -85,B 0,C 180,E1 4037.459,E2 4037.459} C_VEL
LIN {X 0,Y 210.762,Z 1179.487,A -85,B 0,C 180,E1 4031.754,E2 4031.754} C_VEL
LIN {X 0,Y 213.961,Z 1175.798,A -85,B 0,C 180,E1 4026.011,E2 4026.011} C_VEL
LIN {X 0,Y 220.015,Z 1169.886,A -85,B 0,C 180,E1 4019.198,E2 4019.198} C_VEL
LIN {X 0,Y 228.351,Z 1162.183,A -85,B 0,C 180,E1 4012.825,E2 4012.825} C_VEL
LIN {X 0,Y 237.022,Z 1154.514,A -85,B 0,C 180,E1 4007.876,E2 4007.876} C_VEL
LIN {X 0,Y 248.213,Z 1144.677,A -85,B 0,C 180,E1 4002.85,E2 4002.85} C_VEL
LIN {X 0,Y 262.192,Z 1131.944,A -85,B 0,C 180,E1 3997.871,E2 3997.871} C_VEL
LIN {X 0,Y 273.95,Z 1120.814,A -85,B 0,C 180,E1 3994.426,E2 3994.426} C_VEL
LIN {X 0,Y 286.579,Z 1108.304,A -85,B 0,C 180,E1 3991.262,E2 3991.262} C_VEL
LIN {X 0,Y 302.158,Z 1091.865,A -85,B 0,C 180,E1 3987.929,E2 3987.929} C_VEL
LIN {X 0,Y 316.335,Z 1075.577,A -85,B 0,C 180,E1 3985.313,E2 3985.313} C_VEL
LIN {X 0,Y 328.758,Z 1060.276,A -85,B 0,C 180,E1 3983.29,E2 3983.29} C_VEL
LIN {X 0,Y 343.17,Z 1041.091,A -85,B 0,C 180,E1 3981.194,E2 3981.194} C_VEL
LIN {X 0,Y 356.723,Z 1020.854,A -85,B 0,C 180,E1 3979.417,E2 3979.417} C_VEL
LIN {X 0,Y 367.664,Z 1002.94,A -85,B 0,C 180,E1 3978.108,E2 3978.108} C_VEL
LIN {X 0,Y 378.34,Z 983.682,A -85,B 0,C 180,E1 3976.925,E2 3976.925} C_VEL
LIN {X 0,Y 390.92,Z 957.883,A -85,B 0,C 180,E1 3975.637,E2 3975.637} C_VEL
LIN {X 0,Y 399.715,Z 937.062,A -85,B 0,C 180,E1 3974.802,E2 3974.802} C_VEL
LIN {X 0,Y 406.806,Z 917.957,A -85,B 0,C 180,E1 3974.158,E2 3974.158} C_VEL
LIN {X 0,Y 414.17,Z 894.955,A -85,B 0,C 180,E1 3973.517,E2 3973.517} C_VEL
LIN {X 0,Y 421.171,Z 867.679,A -85,B 0,C 180,E1 3972.938,E2 3972.938} C_VEL
LIN {X 0,Y 425.606,Z 845.337,A -85,B 0,C 180,E1 3972.563,E2 3972.563} C_VEL
LIN {X 0,Y 428.976,Z 822.159,A -85,B 0,C 180,E1 3972.219,E2 3972.219} C_VEL
LIN {X 0,Y 446.025,Z 663.222,A -85,B 0,C 180,E1 3970.06,E2 3970.06} C_VEL
LIN {X 0,Y 446.425,Z 658.231,A -85,B 0,C 180,E1 3969.863,E2 3969.863} C_VEL
LIN {X 0,Y 446.983,Z 645.849,A -85,B 0,C 180,E1 3968.906,E2 3968.906} C_VEL
LIN {X 0,Y 447.369,Z 641.541,A -85,B 0,C 180,E1 3968.751,E2 3968.751} C_VEL
LIN {X 0,Y 447.825,Z 637.207,A -85,B 0,C 180,E1 3968.668,E2 3968.668} C_VEL
LIN {X 0,Y 446.61,Z 633.326,A -85,B 0,C 180,E1 3966.427,E2 3966.427} C_VEL
LIN {X 0,Y 445.715,Z 630.127,A -85,B 0,C 180,E1 3963.086,E2 3963.086} C_VEL
LIN {X 0,Y 446.023,Z 630.136,A -85,B 0,C 180,E1 3959.615,E2 3959.615} C_VEL
LIN {X 0,Y 446.525,Z 630.926,A -85,B 0,C 180,E1 3958.203,E2 3958.203} C_VEL
LIN {X 0,Y 448.216,Z 634.65,A -85,B 0,C 180,E1 3955.201,E2 3955.201} C_VEL
LIN {X 0,Y 448.509,Z 635.531,A -85,B 0,C 180,E1 3954.784,E2 3954.784} C_VEL
LIN {X 0,Y 427.213,Z 827.599,A -85,B 0,C 180,E1 3952.121,E2 3952.121} C_VEL
LIN {X 0,Y 422.865,Z 854.276,A -85,B 0,C 180,E1 3951.709,E2 3951.709} C_VEL
LIN {X 0,Y 416.739,Z 880.542,A -85,B 0,C 180,E1 3951.22,E2 3951.22} C_VEL
LIN {X 0,Y 410.86,Z 901.207,A -85,B 0,C 180,E1 3950.733,E2 3950.733} C_VEL
LIN {X 0,Y 403.918,Z 921.997,A -85,B 0,C 180,E1 3950.137,E2 3950.137} C_VEL
LIN {X 0,Y 394.339,Z 946.695,A -85,B 0,C 180,E1 3949.274,E2 3949.274} C_VEL
LIN {X 0,Y 383.545,Z 970.229,A -85,B 0,C 180,E1 3948.245,E2 3948.245} C_VEL
LIN {X 0,Y 373.805,Z 989.192,A -85,B 0,C 180,E1 3947.252,E2 3947.252} C_VEL
LIN {X 0,Y 362.247,Z 1009.522,A -85,B 0,C 180,E1 3945.979,E2 3945.979} C_VEL
LIN {X 0,Y 347.142,Z 1033.179,A -85,B 0,C 180,E1 3944.158,E2 3944.158} C_VEL
LIN {X 0,Y 334.932,Z 1050.461,A -85,B 0,C 180,E1 3942.531,E2 3942.531} C_VEL
LIN {X 0,Y 322.497,Z 1066.731,A -85,B 0,C 180,E1 3940.714,E2 3940.714} C_VEL
LIN {X 0,Y 307.532,Z 1084.953,A -85,B 0,C 180,E1 3938.244,E2 3938.244} C_VEL
LIN {X 0,Y 291.759,Z 1102.51,A -85,B 0,C 180,E1 3935.253,E2 3935.253} C_VEL
LIN {X 0,Y 278.711,Z 1116.161,A -85,B 0,C 180,E1 3932.388,E2 3932.388} C_VEL
LIN {X 0,Y 265.741,Z 1129.087,A -85,B 0,C 180,E1 3929.077,E2 3929.077} C_VEL
LIN {X 0,Y 250.685,Z 1143.497,A -85,B 0,C 180,E1 3924.455,E2 3924.455} C_VEL
LIN {X 0,Y 237.795,Z 1155.286,A -85,B 0,C 180,E1 3919.557,E2 3919.557} C_VEL
LIN {X 0,Y 228.005,Z 1164.244,A -85,B 0,C 180,E1 3914.913,E2 3914.913} C_VEL
LIN {X 0,Y 218.899,Z 1172.762,A -85,B 0,C 180,E1 3909.413,E2 3909.413} C_VEL
LIN {X 0,Y 209.964,Z 1181.626,A -85,B 0,C 180,E1 3901.91,E2 3901.91} C_VEL
LIN {X 0,Y 205.074,Z 1187.108,A -85,B 0,C 180,E1 3895.717,E2 3895.717} C_VEL
LIN {X 0,Y 202.065,Z 1191.208,A -85,B 0,C 180,E1 3889.662,E2 3889.662} C_VEL
LIN {X 0,Y 200.602,Z 1193.973,A -85,B 0,C 180,E1 3884.136,E2 3884.136} C_VEL
LIN {X 0,Y 200.079,Z 1195.77,A -85,B 0,C 180,E1 3878.912,E2 3878.912} C_VEL
LIN {X 0,Y 200.005,Z 1196.743,A -85,B 0,C 180,E1 3874.013,E2 3874.013} C_VEL
LIN {X 0,Y 200.024,Z 1196.979,A -85,B 0,C 180,E1 3868.789,E2 3868.789} C_VEL
LIN {X 0,Y 200.016,Z 1196.343,A -85,B 0,C 180,E1 3863.397,E2 3863.397} C_VEL
LIN {X 0,Y 200.381,Z 1194.559,A -85,B 0,C 180,E1 3857.317,E2 3857.317} C_VEL
LIN {X 0,Y 201.784,Z 1191.666,A -85,B 0,C 180,E1 3851.166,E2 3851.166} C_VEL
LIN {X 0,Y 204.55,Z 1187.728,A -85,B 0,C 180,E1 3845.141,E2 3845.141} C_VEL
LIN {X 0,Y 208.93,Z 1182.649,A -85,B 0,C 180,E1 3839.198,E2 3839.198} C_VEL
LIN {X 0,Y 215.691,Z 1175.797,A -85,B 0,C 180,E1 3832.94,E2 3832.94} C_VEL
LIN {X 0,Y 226.222,Z 1165.85,A -85,B 0,C 180,E1 3826.058,E2 3826.058} C_VEL
LIN {X 0,Y 236.232,Z 1156.627,A -85,B 0,C 180,E1 3821.113,E2 3821.113} C_VEL
LIN {X 0,Y 247.152,Z 1146.589,A -85,B 0,C 180,E1 3816.771,E2 3816.771} C_VEL
LIN {X 0,Y 261.676,Z 1133.025,A -85,B 0,C 180,E1 3812.082,E2 3812.082} C_VEL
LIN {X 0,Y 276.606,Z 1118.172,A -85,B 0,C 180,E1 3808.113,E2 3808.113} C_VEL
LIN {X 0,Y 289.534,Z 1104.714,A -85,B 0,C 180,E1 3805.204,E2 3805.204} C_VEL
LIN {X 0,Y 303.126,Z 1089.752,A -85,B 0,C 180,E1 3802.541,E2 3802.541} C_VEL
LIN {X 0,Y 320.115,Z 1069.544,A -85,B 0,C 180,E1 3799.655,E2 3799.655} C_VEL
LIN {X 0,Y 333.234,Z 1052.5,A -85,B 0,C 180,E1 3797.698,E2 3797.698} C_VEL
LIN {X 0,Y 344.996,Z 1035.986,A -85,B 0,C 180,E1 3796.102,E2 3796.102} C_VEL
LIN {X 0,Y 357.879,Z 1016.324,A -85,B 0,C 180,E1 3794.513,E2 3794.513} C_VEL
LIN {X 0,Y 371.903,Z 992.315,A -85,B 0,C 180,E1 3792.941,E2 3792.941} C_VEL
LIN {X 0,Y 382.144,Z 972.622,A -85,B 0,C 180,E1 3791.882,E2 3791.882} C_VEL
LIN {X 0,Y 391.151,Z 953.327,A -85,B 0,C 180,E1 3791.007,E2 3791.007} C_VEL
LIN {X 0,Y 400.705,Z 930.205,A -85,B 0,C 180,E1 3790.134,E2 3790.134} C_VEL
LIN {X 0,Y 409.653,Z 904.356,A -85,B 0,C 180,E1 3789.358,E2 3789.358} C_VEL
LIN {X 0,Y 415.937,Z 882.675,A -85,B 0,C 180,E1 3788.833,E2 3788.833} C_VEL
LIN {X 0,Y 421.255,Z 860.489,A -85,B 0,C 180,E1 3788.404,E2 3788.404} C_VEL
LIN {X 0,Y 426.376,Z 832.158,A -85,B 0,C 180,E1 3787.952,E2 3787.952} C_VEL
LIN {X 0,Y 432.563,Z 778.434,A -85,B 0,C 180,E1 3787.192,E2 3787.192} C_VEL
LIN {X 0,Y 448.324,Z 635.164,A -85,B 0,C 180,E1 3785.215,E2 3785.215} C_VEL
LIN {X 0,Y 447.177,Z 632.788,A -85,B 0,C 180,E1 3783.59,E2 3783.59} C_VEL
LIN {X 0,Y 446.092,Z 630.253,A -85,B 0,C 180,E1 3781.284,E2 3781.284} C_VEL
LIN {X 0,Y 445.4,Z 629.714,A -85,B 0,C 180,E1 3777.942,E2 3777.942} C_VEL
LIN {X 0,Y 445.541,Z 630.325,A -85,B 0,C 180,E1 3776.14,E2 3776.14} C_VEL
LIN {X 0,Y 446.611,Z 634.034,A -85,B 0,C 180,E1 3772.862,E2 3772.862} C_VEL
LIN {X 0,Y 447.574,Z 637.087,A -85,B 0,C 180,E1 3771.213,E2 3771.213} C_VEL
LIN {X 0,Y 426.467,Z 828.966,A -85,B 0,C 180,E1 3768.648,E2 3768.648} C_VEL
LIN {X 0,Y 422.045,Z 855.876,A -85,B 0,C 180,E1 3768.242,E2 3768.242} C_VEL
LIN {X 0,Y 416.136,Z 881.19,A -85,B 0,C 180,E1 3767.776,E2 3767.776} C_VEL
LIN {X 0,Y 410.229,Z 901.848,A -85,B 0,C 180,E1 3767.307,E2 3767.307} C_VEL
LIN {X 0,Y 402.285,Z 925.369,A -85,B 0,C 180,E1 3766.635,E2 3766.635} C_VEL
LIN {X 0,Y 392.065,Z 950.616,A -85,B 0,C 180,E1 3765.722,E2 3765.722} C_VEL
LIN {X 0,Y 382.783,Z 970.552,A -85,B 0,C 180,E1 3764.837,E2 3764.837} C_VEL
LIN {X 0,Y 372.716,Z 989.851,A -85,B 0,C 180,E1 3763.823,E2 3763.823} C_VEL
LIN {X 0,Y 359.176,Z 1013.002,A -85,B 0,C 180,E1 3762.336,E2 3762.336} C_VEL
LIN {X 0,Y 346.243,Z 1032.568,A -85,B 0,C 180,E1 3760.779,E2 3760.779} C_VEL
LIN {X 0,Y 334.267,Z 1049.164,A -85,B 0,C 180,E1 3759.191,E2 3759.191} C_VEL
LIN {X 0,Y 320.562,Z 1066.659,A -85,B 0,C 180,E1 3757.178,E2 3757.178} C_VEL
LIN {X 0,Y 304.591,Z 1085.146,A -85,B 0,C 180,E1 3754.521,E2 3754.521} C_VEL
LIN {X 0,Y 291.886,Z 1098.762,A -85,B 0,C 180,E1 3752.105,E2 3752.105} C_VEL
LIN {X 0,Y 279.035,Z 1111.709,A -85,B 0,C 180,E1 3749.318,E2 3749.318} C_VEL
LIN {X 0,Y 263.641,Z 1126.36,A -85,B 0,C 180,E1 3745.386,E2 3745.386} C_VEL
LIN {X 0,Y 249.545,Z 1138.831,A -85,B 0,C 180,E1 3741.017,E2 3741.017} C_VEL
LIN {X 0,Y 238.521,Z 1148.306,A -85,B 0,C 180,E1 3736.837,E2 3736.837} C_VEL
LIN {X 0,Y 226.532,Z 1158.511,A -85,B 0,C 180,E1 3731.123,E2 3731.123} C_VEL
LIN {X 0,Y 216.725,Z 1166.715,A -85,B 0,C 180,E1 3724.896,E2 3724.896} C_VEL
LIN {X 0,Y 210.306,Z 1172.385,A -85,B 0,C 180,E1 3719.322,E2 3719.322} C_VEL
LIN {X 0,Y 205.396,Z 1177.138,A -85,B 0,C 180,E1 3713.224,E2 3713.224} C_VEL
LIN {X 0,Y 201.762,Z 1181.364,A -85,B 0,C 180,E1 3705.523,E2 3705.523} C_VEL
LIN {X 0,Y 200.426,Z 1183.518,A -85,B 0,C 180,E1 3698.962,E2 3698.962} C_VEL
LIN {X 0,Y 200.078,Z 1184.454,A -85,B 0,C 180,E1 3693.439,E2 3693.439} C_VEL
LIN {X 0,Y 200.062,Z 1184.591,A -85,B 0,C 180,E1 3688.282,E2 3688.282} C_VEL
LIN {X 0,Y 200.247,Z 1183.948,A -85,B 0,C 180,E1 3682.83,E2 3682.83} C_VEL
LIN {X 0,Y 201.044,Z 1182.383,A -85,B 0,C 180,E1 3677.068,E2 3677.068} C_VEL
LIN {X 0,Y 203.031,Z 1179.74,A -85,B 0,C 180,E1 3671.033,E2 3671.033} C_VEL
LIN {X 0,Y 206.491,Z 1176.051,A -85,B 0,C 180,E1 3665.086,E2 3665.086} C_VEL
LIN {X 0,Y 212.773,Z 1170.306,A -85,B 0,C 180,E1 3658.244,E2 3658.244} C_VEL
LIN {X 0,Y 221.827,Z 1162.441,A -85,B 0,C 180,E1 3651.536,E2 3651.536} C_VEL
LIN {X 0,Y 230.947,Z 1154.774,A -85,B 0,C 180,E1 3646.498,E2 3646.498} C_VEL
LIN {X 0,Y 242.117,Z 1145.384,A -85,B 0,C 180,E1 3641.628,E2 3641.628} C_VEL
LIN {X 0,Y 256.641,Z 1132.722,A -85,B 0,C 180,E1 3636.591,E2 3636.591} C_VEL
LIN {X 0,Y 269.37,Z 1121.086,A -85,B 0,C 180,E1 3632.978,E2 3632.978} C_VEL
LIN {X 0,Y 282.391,Z 1108.579,A -85,B 0,C 180,E1 3629.833,E2 3629.833} C_VEL
LIN {X 0,Y 298.401,Z 1092.155,A -85,B 0,C 180,E1 3626.536,E2 3626.536} C_VEL
LIN {X 0,Y 313.111,Z 1075.655,A -85,B 0,C 180,E1 3623.927,E2 3623.927} C_VEL
LIN {X 0,Y 326.011,Z 1060.094,A -85,B 0,C 180,E1 3621.911,E2 3621.911} C_VEL
LIN {X 0,Y 340.728,Z 1040.849,A -85,B 0,C 180,E1 3619.862,E2 3619.862} C_VEL
LIN {X 0,Y 354.553,Z 1020.523,A -85,B 0,C 180,E1 3618.127,E2 3618.127} C_VEL
LIN {X 0,Y 365.236,Z 1003.321,A -85,B 0,C 180,E1 3616.904,E2 3616.904} C_VEL
LIN {X 0,Y 376.074,Z 984.092,A -85,B 0,C 180,E1 3615.751,E2 3615.751} C_VEL
LIN {X 0,Y 388.393,Z 959.368,A -85,B 0,C 180,E1 3614.542,E2 3614.542} C_VEL
LIN {X 0,Y 397.746,Z 937.609,A -85,B 0,C 180,E1 3613.687,E2 3613.687} C_VEL
LIN {X 0,Y 404.927,Z 918.577,A -85,B 0,C 180,E1 3613.063,E2 3613.063} C_VEL
LIN {X 0,Y 412.108,Z 896.549,A -85,B 0,C 180,E1 3612.462,E2 3612.462} C_VEL
LIN {X 0,Y 419.578,Z 868.184,A -85,B 0,C 180,E1 3611.872,E2 3611.872} C_VEL
LIN {X 0,Y 424.15,Z 845.5,A -85,B 0,C 180,E1 3611.501,E2 3611.501} C_VEL
LIN {X 0,Y 427.555,Z 822.509,A -85,B 0,C 180,E1 3611.166,E2 3611.166} C_VEL
LIN {X 0,Y 447.369,Z 641.541,A -85,B 0,C 180,E1 3608.751,E2 3608.751} C_VEL
LIN {X 0,Y 447.455,Z 639.621,A -85,B 0,C 180,E1 3608.587,E2 3608.587} C_VEL
LIN {X 0,Y 447.266,Z 638.442,A -85,B 0,C 180,E1 3608.204,E2 3608.204} C_VEL
LIN {X 0,Y 446.75,Z 638.476,A -85,B 0,C 180,E1 3607.563,E2 3607.563} C_VEL
LIN {X 0,Y 445.559,Z 640.652,A -85,B 0,C 180,E1 3606.158,E2 3606.158} C_VEL
LIN {X 0,Y 445.313,Z 640.612,A -85,B 0,C 180,E1 3605.684,E2 3605.684} C_VEL
LIN {X 0,Y 444.723,Z 638.043,A -85,B 0,C 180,E1 3602.964,E2 3602.964} C_VEL
LIN {X 0,Y 445.08,Z 638.118,A -85,B 0,C 180,E1 3599.485,E2 3599.485} C_VEL
LIN {X 0,Y 445.532,Z 638.962,A -85,B 0,C 180,E1 3598.199,E2 3598.199} C_VEL
LIN {X 0,Y 446.83,Z 642.024,A -85,B 0,C 180,E1 3595.716,E2 3595.716} C_VEL
LIN {X 0,Y 425.924,Z 827.676,A -85,B 0,C 180,E1 3593.185,E2 3593.185} C_VEL
LIN {X 0,Y 421.512,Z 854.403,A -85,B 0,C 180,E1 3592.781,E2 3592.781} C_VEL
LIN {X 0,Y 415.342,Z 880.556,A -85,B 0,C 180,E1 3592.311,E2 3592.311} C_VEL
LIN {X 0,Y 409.391,Z 901.233,A -85,B 0,C 180,E1 3591.839,E2 3591.839} C_VEL
LIN {X 0,Y 402.6,Z 921.365,A -85,B 0,C 180,E1 3591.282,E2 3591.282} C_VEL
LIN {X 0,Y 392.898,Z 946.182,A -85,B 0,C 180,E1 3590.447,E2 3590.447} C_VEL
LIN {X 0,Y 381.795,Z 970.093,A -85,B 0,C 180,E1 3589.436,E2 3589.436} C_VEL
LIN {X 0,Y 371.949,Z 988.996,A -85,B 0,C 180,E1 3588.477,E2 3588.477} C_VEL
LIN {X 0,Y 360.777,Z 1008.384,A -85,B 0,C 180,E1 3587.303,E2 3587.303} C_VEL
LIN {X 0,Y 345.839,Z 1031.597,A -85,B 0,C 180,E1 3585.588,E2 3585.588} C_VEL
LIN {X 0,Y 332.499,Z 1050.159,A -85,B 0,C 180,E1 3583.9,E2 3583.9} C_VEL
LIN {X 0,Y 320.156,Z 1066.007,A -85,B 0,C 180,E1 3582.177,E2 3582.177} C_VEL
LIN {X 0,Y 306.391,Z 1082.441,A -85,B 0,C 180,E1 3580.027,E2 3580.027} C_VEL
LIN {X 0,Y 289.1,Z 1101.434,A -85,B 0,C 180,E1 3576.923,E2 3576.923} C_VEL
LIN {X 0,Y 274.899,Z 1115.874,A -85,B 0,C 180,E1 3573.948,E2 3573.948} C_VEL
LIN {X 0,Y 261.494,Z 1128.806,A -85,B 0,C 180,E1 3570.668,E2 3570.668} C_VEL
LIN {X 0,Y 245.858,Z 1143.226,A -85,B 0,C 180,E1 3566.061,E2 3566.061} C_VEL
LIN {X 0,Y 232.404,Z 1155.017,A -85,B 0,C 180,E1 3561.143,E2 3561.143} C_VEL
LIN {X 0,Y 221.623,Z 1164.398,A -85,B 0,C 180,E1 3556.207,E2 3556.207} C_VEL
LIN {X 0,Y 211.286,Z 1173.598,A -85,B 0,C 180,E1 3550.06,E2 3550.06} C_VEL
LIN {X 0,Y 202.622,Z 1181.633,A -85,B 0,C 180,E1 3542.875,E2 3542.875} C_VEL
LIN {X 0,Y 197.423,Z 1187.069,A -85,B 0,C 180,E1 3536.467,E2 3536.467} C_VEL
LIN {X 0,Y 194.208,Z 1191.124,A -85,B 0,C 180,E1 3530.178,E2 3530.178} C_VEL
LIN {X 0,Y 192.643,Z 1193.842,A -85,B 0,C 180,E1 3524.426,E2 3524.426} C_VEL
LIN {X 0,Y 192.083,Z 1195.594,A -85,B 0,C 180,E1 3518.984,E2 3518.984} C_VEL
LIN {X 0,Y 192.009,Z 1196.521,A -85,B 0,C 180,E1 3513.881,E2 3513.881} C_VEL
LIN {X 0,Y 192.027,Z 1196.731,A -85,B 0,C 180,E1 3508.734,E2 3508.734} C_VEL
LIN {X 0,Y 192.022,Z 1196.094,A -85,B 0,C 180,E1 3503.121,E2 3503.121} C_VEL
LIN {X 0,Y 192.449,Z 1194.307,A -85,B 0,C 180,E1 3496.784,E2 3496.784} C_VEL
LIN {X 0,Y 193.992,Z 1191.435,A -85,B 0,C 180,E1 3490.425,E2 3490.425} C_VEL
LIN {X 0,Y 197.046,Z 1187.469,A -85,B 0,C 180,E1 3484.125,E2 3484.125} C_VEL
LIN {X 0,Y 201.902,Z 1182.286,A -85,B 0,C 180,E1 3477.871,E2 3477.871} C_VEL
LIN {X 0,Y 209.403,Z 1175.217,A -85,B 0,C 180,E1 3471.28,E2 3471.28} C_VEL
LIN {X 0,Y 220.214,Z 1165.58,A -85,B 0,C 180,E1 3464.532,E2 3464.532} C_VEL
LIN {X 0,Y 230.76,Z 1156.356,A -85,B 0,C 180,E1 3459.531,E2 3459.531} C_VEL
LIN {X 0,Y 242.186,Z 1146.313,A -85,B 0,C 180,E1 3455.169,E2 3455.169} C_VEL
LIN {X 0,Y 256.787,Z 1133.185,A -85,B 0,C 180,E1 3450.623,E2 3450.623} C_VEL
LIN {X 0,Y 272.723,Z 1117.882,A -85,B 0,C 180,E1 3446.546,E2 3446.546} C_VEL
LIN {X 0,Y 286.044,Z 1104.417,A -85,B 0,C 180,E1 3443.675,E2 3443.675} C_VEL
LIN {X 0,Y 300.003,Z 1089.449,A -85,B 0,C 180,E1 3441.058,E2 3441.058} C_VEL
LIN {X 0,Y 317.395,Z 1069.217,A -85,B 0,C 180,E1 3438.23,E2 3438.23} C_VEL
LIN {X 0,Y 330.734,Z 1052.239,A -85,B 0,C 180,E1 3436.33,E2 3436.33} C_VEL
LIN {X 0,Y 342.786,Z 1035.629,A -85,B 0,C 180,E1 3434.769,E2 3434.769} C_VEL
LIN {X 0,Y 355.895,Z 1015.948,A -85,B 0,C 180,E1 3433.223,E2 3433.223} C_VEL
LIN {X 0,Y 369.694,Z 992.703,A -85,B 0,C 180,E1 3431.742,E2 3431.742} C_VEL
LIN {X 0,Y 380.119,Z 972.988,A -85,B 0,C 180,E1 3430.711,E2 3430.711} C_VEL
LIN {X 0,Y 389.278,Z 953.676,A -85,B 0,C 180,E1 3429.859,E2 3429.859} C_VEL
LIN {X 0,Y 398.884,Z 930.774,A -85,B 0,C 180,E1 3429.018,E2 3429.018} C_VEL
LIN {X 0,Y 408.174,Z 904.359,A -85,B 0,C 180,E1 3428.248,E2 3428.248} C_VEL
LIN {X 0,Y 414.61,Z 882.382,A -85,B 0,C 180,E1 3427.734,E2 3427.734} C_VEL
LIN {X 0,Y 420.056,Z 859.822,A -85,B 0,C 180,E1 3427.315,E2 3427.315} C_VEL
LIN {X 0,Y 425.354,Z 830.115,A -85,B 0,C 180,E1 3426.856,E2 3426.856} C_VEL
LIN {X 0,Y 433.901,Z 755.615,A -85,B 0,C 180,E1 3425.825,E2 3425.825} C_VEL
LIN {X 0,Y 446.64,Z 641.598,A -85,B 0,C 180,E1 3424.269,E2 3424.269} C_VEL
LIN {X 0,Y 445.061,Z 638.15,A -85,B 0,C 180,E1 3421.159,E2 3421.159} C_VEL
LIN {X 0,Y 444.426,Z 637.656,A -85,B 0,C 180,E1 3417.937,E2 3417.937} C_VEL
LIN {X 0,Y 444.545,Z 638.21,A -85,B 0,C 180,E1 3416.26,E2 3416.26} C_VEL
LIN {X 0,Y 445.529,Z 641.844,A -85,B 0,C 180,E1 3413.039,E2 3413.039} C_VEL
LIN {X 0,Y 445.971,Z 643.515,A -85,B 0,C 180,E1 3412.153,E2 3412.153} C_VEL
LIN {X 0,Y 425.226,Z 828.888,A -85,B 0,C 180,E1 3409.716,E2 3409.716} C_VEL
LIN {X 0,Y 420.751,Z 855.794,A -85,B 0,C 180,E1 3409.32,E2 3409.32} C_VEL
LIN {X 0,Y 414.787,Z 881.069,A -85,B 0,C 180,E1 3408.871,E2 3408.871} C_VEL
LIN {X 0,Y 408.78,Z 901.845,A -85,B 0,C 180,E1 3408.416,E2 3408.416} C_VEL
LIN {X 0,Y 401.027,Z 924.569,A -85,B 0,C 180,E1 3407.789,E2 3407.789} C_VEL
LIN {X 0,Y 390.619,Z 950.124,A -85,B 0,C 180,E1 3406.901,E2 3406.901} C_VEL
LIN {X 0,Y 381.206,Z 970.12,A -85,B 0,C 180,E1 3406.046,E2 3406.046} C_VEL
LIN {X 0,Y 371.432,Z 988.668,A -85,B 0,C 180,E1 3405.109,E2 3405.109} C_VEL
LIN {X 0,Y 358.3,Z 1011.085,A -85,B 0,C 180,E1 3403.735,E2 3403.735} C_VEL
LIN {X 0,Y 344.101,Z 1032.288,A -85,B 0,C 180,E1 3402.109,E2 3402.109} C_VEL
LIN {X 0,Y 331.883,Z 1048.943,A -85,B 0,C 180,E1 3400.561,E2 3400.561} C_VEL
LIN {X 0,Y 318.701,Z 1065.476,A -85,B 0,C 180,E1 3398.717,E2 3398.717} C_VEL
LIN {X 0,Y 301.941,Z 1084.606,A -85,B 0,C 180,E1 3396.061,E2 3396.061} C_VEL
LIN {X 0,Y 288.134,Z 1099.049,A -85,B 0,C 180,E1 3393.549,E2 3393.549} C_VEL
LIN {X 0,Y 274.923,Z 1111.99,A -85,B 0,C 180,E1 3390.794,E2 3390.794} C_VEL
LIN {X 0,Y 259.043,Z 1126.629,A -85,B 0,C 180,E1 3386.888,E2 3386.888} C_VEL
LIN {X 0,Y 244.43,Z 1139.097,A -85,B 0,C 180,E1 3382.523,E2 3382.523} C_VEL
LIN {X 0,Y 232.776,Z 1148.706,A -85,B 0,C 180,E1 3378.256,E2 3378.256} C_VEL
LIN {X 0,Y 220.374,Z 1158.771,A -85,B 0,C 180,E1 3372.536,E2 3372.536} C_VEL
LIN {X 0,Y 210.011,Z 1166.972,A -85,B 0,C 180,E1 3366.184,E2 3366.184} C_VEL
LIN {X 0,Y 203.17,Z 1172.642,A -85,B 0,C 180,E1 3360.458,E2 3360.458} C_VEL
LIN {X 0,Y 197.896,Z 1177.393,A -85,B 0,C 180,E1 3354.159,E2 3354.159} C_VEL
LIN {X 0,Y 193.946,Z 1181.615,A -85,B 0,C 180,E1 3346.165,E2 3346.165} C_VEL
LIN {X 0,Y 192.506,Z 1183.718,A -85,B 0,C 180,E1 3339.568,E2 3339.568} C_VEL
LIN {X 0,Y 192.093,Z 1184.68,A -85,B 0,C 180,E1 3333.881,E2 3333.881} C_VEL
LIN {X 0,Y 192.066,Z 1184.844,A -85,B 0,C 180,E1 3328.287,E2 3328.287} C_VEL
LIN {X 0,Y 192.274,Z 1184.196,A -85,B 0,C 180,E1 3322.531,E2 3322.531} C_VEL
LIN {X 0,Y 193.158,Z 1182.633,A -85,B 0,C 180,E1 3316.53,E2 3316.53} C_VEL
LIN {X 0,Y 195.331,Z 1179.991,A -85,B 0,C 180,E1 3310.255,E2 3310.255} C_VEL
LIN {X 0,Y 199.156,Z 1176.234,A -85,B 0,C 180,E1 3303.988,E2 3303.988} C_VEL
LIN {X 0,Y 206.135,Z 1170.314,A -85,B 0,C 180,E1 3296.763,E2 3296.763} C_VEL
LIN {X 0,Y 215.42,Z 1162.699,A -85,B 0,C 180,E1 3290.169,E2 3290.169} C_VEL
LIN {X 0,Y 225.015,Z 1155.032,A -85,B 0,C 180,E1 3285.047,E2 3285.047} C_VEL
LIN {X 0,Y 237.272,Z 1145.197,A -85,B 0,C 180,E1 3279.92,E2 3279.92} C_VEL
LIN {X 0,Y 252.38,Z 1132.478,A -85,B 0,C 180,E1 3274.907,E2 3274.907} C_VEL
LIN {X 0,Y 264.968,Z 1121.356,A -85,B 0,C 180,E1 3271.48,E2 3271.48} C_VEL
LIN {X 0,Y 278.385,Z 1108.852,A -85,B 0,C 180,E1 3268.363,E2 3268.363} C_VEL
LIN {X 0,Y 295.112,Z 1092.133,A -85,B 0,C 180,E1 3265.057,E2 3265.057} C_VEL
LIN {X 0,Y 309.69,Z 1076.172,A -85,B 0,C 180,E1 3262.574,E2 3262.574} C_VEL
LIN {X 0,Y 323.011,Z 1060.455,A -85,B 0,C 180,E1 3260.574,E2 3260.574} C_VEL
LIN {X 0,Y 338.198,Z 1040.978,A -85,B 0,C 180,E1 3258.547,E2 3258.547} C_VEL
LIN {X 0,Y 352.117,Z 1020.881,A -85,B 0,C 180,E1 3256.874,E2 3256.874} C_VEL
LIN {X 0,Y 363.409,Z 1002.974,A -85,B 0,C 180,E1 3255.639,E2 3255.639} C_VEL
LIN {X 0,Y 374.369,Z 983.778,A -85,B 0,C 180,E1 3254.525,E2 3254.525} C_VEL
LIN {X 0,Y 387.353,Z 957.869,A -85,B 0,C 180,E1 3253.308,E2 3253.308} C_VEL
LIN {X 0,Y 396.38,Z 937.039,A -85,B 0,C 180,E1 3252.523,E2 3252.523} C_VEL
LIN {X 0,Y 403.656,Z 917.923,A -85,B 0,C 180,E1 3251.922,E2 3251.922} C_VEL
LIN {X 0,Y 411.361,Z 894.398,A -85,B 0,C 180,E1 3251.309,E2 3251.309} C_VEL
LIN {X 0,Y 418.418,Z 867.395,A -85,B 0,C 180,E1 3250.775,E2 3250.775} C_VEL
LIN {X 0,Y 422.955,Z 845.018,A -85,B 0,C 180,E1 3250.422,E2 3250.422} C_VEL
LIN {X 0,Y 426.475,Z 821.364,A -85,B 0,C 180,E1 3250.085,E2 3250.085} C_VEL
LIN {X 0,Y 446.273,Z 643.497,A -85,B 0,C 180,E1 3247.744,E2 3247.744} C_VEL
LIN {X 0,Y 445.41,Z 640.844,A -85,B 0,C 180,E1 3245.927,E2 3245.927} C_VEL
LIN {X 0,Y 445.313,Z 640.612,A -85,B 0,C 180,E1 3245.684,E2 3245.684} C_VEL
LIN {X 0,Y 444.868,Z 640.672,A -85,B 0,C 180,E1 3244.684,E2 3244.684} C_VEL
LIN {X 0,Y 444.015,Z 643.738,A -85,B 0,C 180,E1 3242.847,E2 3242.847} C_VEL
LIN {X 0,Y 443.732,Z 645.653,A -85,B 0,C 180,E1 3241.487,E2 3241.487} C_VEL
LIN {X 0,Y 443.751,Z 645.776,A -85,B 0,C 180,E1 3241.124,E2 3241.124} C_VEL
LIN {X 0,Y 444.408,Z 646.519,A -85,B 0,C 180,E1 3238.582,E2 3238.582} C_VEL
LIN {X 0,Y 445.25,Z 648.931,A -85,B 0,C 180,E1 3236.651,E2 3236.651} C_VEL
LIN {X 0,Y 424.768,Z 827.874,A -85,B 0,C 180,E1 3234.253,E2 3234.253} C_VEL
LIN {X 0,Y 420.285,Z 854.634,A -85,B 0,C 180,E1 3233.858,E2 3233.858} C_VEL
LIN {X 0,Y 414.062,Z 880.697,A -85,B 0,C 180,E1 3233.405,E2 3233.405} C_VEL
LIN {X 0,Y 407.797,Z 902.141,A -85,B 0,C 180,E1 3232.931,E2 3232.931} C_VEL
LIN {X 0,Y 400.505,Z 923.329,A -85,B 0,C 180,E1 3232.358,E2 3232.358} C_VEL
LIN {X 0,Y 389.757,Z 949.757,A -85,B 0,C 180,E1 3231.474,E2 3231.474} C_VEL
LIN {X 0,Y 379.615,Z 971.137,A -85,B 0,C 180,E1 3230.585,E2 3230.585} C_VEL
LIN {X 0,Y 369.478,Z 990.219,A -85,B 0,C 180,E1 3229.638,E2 3229.638} C_VEL
LIN {X 0,Y 356.352,Z 1012.46,A -85,B 0,C 180,E1 3228.305,E2 3228.305} C_VEL
LIN {X 0,Y 341.657,Z 1034.338,A -85,B 0,C 180,E1 3226.673,E2 3226.673} C_VEL
LIN {X 0,Y 329.419,Z 1050.957,A -85,B 0,C 180,E1 3225.179,E2 3225.179} C_VEL
LIN {X 0,Y 316.148,Z 1067.578,A -85,B 0,C 180,E1 3223.393,E2 3223.393} C_VEL
LIN {X 0,Y 299.535,Z 1086.75,A -85,B 0,C 180,E1 3220.852,E2 3220.852} C_VEL
LIN {X 0,Y 283.551,Z 1103.506,A -85,B 0,C 180,E1 3218.033,E2 3218.033} C_VEL
LIN {X 0,Y 269.804,Z 1117.025,A -85,B 0,C 180,E1 3215.223,E2 3215.223} C_VEL
LIN {X 0,Y 253.965,Z 1131.78,A -85,B 0,C 180,E1 3211.397,E2 3211.397} C_VEL
LIN {X 0,Y 238.047,Z 1145.607,A -85,B 0,C 180,E1 3206.705,E2 3206.705} C_VEL
LIN {X 0,Y 226.05,Z 1155.697,A -85,B 0,C 180,E1 3202.35,E2 3202.35} C_VEL
LIN {X 0,Y 214.866,Z 1164.969,A -85,B 0,C 180,E1 3197.328,E2 3197.328} C_VEL
LIN {X 0,Y 202.907,Z 1175.011,A -85,B 0,C 180,E1 3190.205,E2 3190.205} C_VEL
LIN {X 0,Y 195.046,Z 1181.906,A -85,B 0,C 180,E1 3183.617,E2 3183.617} C_VEL
LIN {X 0,Y 189.807,Z 1187.028,A -85,B 0,C 180,E1 3177.277,E2 3177.277} C_VEL
LIN {X 0,Y 186.37,Z 1191.038,A -85,B 0,C 180,E1 3170.737,E2 3170.737} C_VEL
LIN {X 0,Y 184.631,Z 1193.832,A -85,B 0,C 180,E1 3164.424,E2 3164.424} C_VEL
LIN {X 0,Y 184.057,Z 1195.638,A -85,B 0,C 180,E1 3158.119,E2 3158.119} C_VEL
LIN {X 0,Y 184.02,Z 1196.373,A -85,B 0,C 180,E1 3152.802,E2 3152.802} C_VEL
LIN {X 0,Y 184.027,Z 1196.442,A -85,B 0,C 180,E1 3148.131,E2 3148.131} C_VEL
LIN {X 0,Y 184.044,Z 1195.772,A -85,B 0,C 180,E1 3142.507,E2 3142.507} C_VEL
LIN {X 0,Y 184.578,Z 1193.933,A -85,B 0,C 180,E1 3135.89,E2 3135.89} C_VEL
LIN {X 0,Y 186.249,Z 1191.178,A -85,B 0,C 180,E1 3129.576,E2 3129.576} C_VEL
LIN {X 0,Y 189.604,Z 1187.211,A -85,B 0,C 180,E1 3123.029,E2 3123.029} C_VEL
LIN {X 0,Y 194.753,Z 1182.128,A -85,B 0,C 180,E1 3116.677,E2 3116.677} C_VEL
LIN {X 0,Y 202.517,Z 1175.27,A -85,B 0,C 180,E1 3110.07,E2 3110.07} C_VEL
LIN {X 0,Y 214.37,Z 1165.311,A -85,B 0,C 180,E1 3102.921,E2 3102.921} C_VEL
LIN {X 0,Y 225.477,Z 1156.084,A -85,B 0,C 180,E1 3097.875,E2 3097.875} C_VEL
LIN {X 0,Y 237.497,Z 1145.969,A -85,B 0,C 180,E1 3093.472,E2 3093.472} C_VEL
LIN {X 0,Y 252.579,Z 1132.907,A -85,B 0,C 180,E1 3088.97,E2 3088.97} C_VEL
LIN {X 0,Y 269.053,Z 1117.592,A -85,B 0,C 180,E1 3084.936,E2 3084.936} C_VEL
LIN {X 0,Y 282.763,Z 1104.121,A -85,B 0,C 180,E1 3082.11,E2 3082.11} C_VEL
LIN {X 0,Y 297.086,Z 1089.146,A -85,B 0,C 180,E1 3079.545,E2 3079.545} C_VEL
LIN {X 0,Y 315.296,Z 1068.375,A -85,B 0,C 180,E1 3076.721,E2 3076.721} C_VEL
LIN {X 0,Y 328.713,Z 1051.601,A -85,B 0,C 180,E1 3074.903,E2 3074.903} C_VEL
LIN {X 0,Y 341.206,Z 1034.656,A -85,B 0,C 180,E1 3073.368,E2 3073.368} C_VEL
LIN {X 0,Y 355.445,Z 1013.54,A -85,B 0,C 180,E1 3071.78,E2 3071.78} C_VEL
LIN {X 0,Y 369.014,Z 990.627,A -85,B 0,C 180,E1 3070.396,E2 3070.396} C_VEL
LIN {X 0,Y 379.101,Z 971.683,A -85,B 0,C 180,E1 3069.45,E2 3069.45} C_VEL
LIN {X 0,Y 388.355,Z 952.296,A -85,B 0,C 180,E1 3068.633,E2 3068.633} C_VEL
LIN {X 0,Y 398.625,Z 927.857,A -85,B 0,C 180,E1 3067.782,E2 3067.782} C_VEL
LIN {X 0,Y 407.32,Z 902.867,A -85,B 0,C 180,E1 3067.094,E2 3067.094} C_VEL
LIN {X 0,Y 413.65,Z 881.297,A -85,B 0,C 180,E1 3066.613,E2 3066.613} C_VEL
LIN {X 0,Y 419.617,Z 856.466,A -85,B 0,C 180,E1 3066.176,E2 3066.176} C_VEL
LIN {X 0,Y 424.393,Z 828.774,A -85,B 0,C 180,E1 3065.765,E2 3065.765} C_VEL
LIN {X 0,Y 437.98,Z 710.456,A -85,B 0,C 180,E1 3064.169,E2 3064.169} C_VEL
LIN {X 0,Y 445.022,Z 648.5,A -85,B 0,C 180,E1 3063.317,E2 3063.317} C_VEL
LIN {X 0,Y 444.012,Z 646.026,A -85,B 0,C 180,E1 3060.977,E2 3060.977} C_VEL
LIN {X 0,Y 443.45,Z 645.62,A -85,B 0,C 180,E1 3057.803,E2 3057.803} C_VEL
LIN {X 0,Y 443.562,Z 646.237,A -85,B 0,C 180,E1 3056.252,E2 3056.252} C_VEL
LIN {X 0,Y 444.48,Z 649.762,A -85,B 0,C 180,E1 3053.152,E2 3053.152} C_VEL
LIN {X 0,Y 444.467,Z 650.167,A -85,B 0,C 180,E1 3053.096,E2 3053.096} C_VEL
LIN {X 0,Y 424.131,Z 828.823,A -85,B 0,C 180,E1 3050.789,E2 3050.789} C_VEL
LIN {X 0,Y 419.614,Z 855.676,A -85,B 0,C 180,E1 3050.405,E2 3050.405} C_VEL
LIN {X 0,Y 413.583,Z 880.975,A -85,B 0,C 180,E1 3049.971,E2 3049.971} C_VEL
LIN {X 0,Y 407.612,Z 901.439,A -85,B 0,C 180,E1 3049.541,E2 3049.541} C_VEL
LIN {X 0,Y 399.968,Z 923.669,A -85,B 0,C 180,E1 3048.952,E2 3048.952} C_VEL
LIN {X 0,Y 389.34,Z 949.632,A -85,B 0,C 180,E1 3048.088,E2 3048.088} C_VEL
LIN {X 0,Y 379.8,Z 969.688,A -85,B 0,C 180,E1 3047.264,E2 3047.264} C_VEL
LIN {X 0,Y 369.892,Z 988.287,A -85,B 0,C 180,E1 3046.359,E2 3046.359} C_VEL
LIN {X 0,Y 357.885,Z 1008.579,A -85,B 0,C 180,E1 3045.167,E2 3045.167} C_VEL
LIN {X 0,Y 343.001,Z 1030.83,A -85,B 0,C 180,E1 3043.55,E2 3043.55} C_VEL
LIN {X 0,Y 330.499,Z 1047.683,A -85,B 0,C 180,E1 3042.05,E2 3042.05} C_VEL
LIN {X 0,Y 317.487,Z 1063.793,A -85,B 0,C 180,E1 3040.332,E2 3040.332} C_VEL
LIN {X 0,Y 301.121,Z 1082.404,A -85,B 0,C 180,E1 3037.885,E2 3037.885} C_VEL
LIN {X 0,Y 285.339,Z 1098.576,A -85,B 0,C 180,E1 3035.174,E2 3035.174} C_VEL
LIN {X 0,Y 271.735,Z 1111.582,A -85,B 0,C 180,E1 3032.473,E2 3032.473} C_VEL
LIN {X 0,Y 256.696,Z 1125.092,A -85,B 0,C 180,E1 3028.975,E2 3028.975} C_VEL
LIN {X 0,Y 240.462,Z 1138.591,A -85,B 0,C 180,E1 3024.398,E2 3024.398} C_VEL
LIN {X 0,Y 228.092,Z 1148.387,A -85,B 0,C 180,E1 3020.098,E2 3020.098} C_VEL
LIN {X 0,Y 216.219,Z 1157.544,A -85,B 0,C 180,E1 3014.965,E2 3014.965} C_VEL
LIN {X 0,Y 204.189,Z 1166.645,A -85,B 0,C 180,E1 3008.098,E2 3008.098} C_VEL
LIN {X 0,Y 196.425,Z 1172.653,A -85,B 0,C 180,E1 3001.965,E2 3001.965} C_VEL
LIN {X 0,Y 190.796,Z 1177.327,A -85,B 0,C 180,E1 2995.659,E2 2995.659} C_VEL
LIN {X 0,Y 186.498,Z 1181.534,A -85,B 0,C 180,E1 2987.795,E2 2987.795} C_VEL
LIN {X 0,Y 184.558,Z 1183.967,A -85,B 0,C 180,E1 2979.984,E2 2979.984} C_VEL
LIN {X 0,Y 184.101,Z 1184.928,A -85,B 0,C 180,E1 2974.049,E2 2974.049} C_VEL
LIN {X 0,Y 184.07,Z 1185.091,A -85,B 0,C 180,E1 2968.213,E2 2968.213} C_VEL
LIN {X 0,Y 184.304,Z 1184.445,A -85,B 0,C 180,E1 2962.206,E2 2962.206} C_VEL
LIN {X 0,Y 185.286,Z 1182.882,A -85,B 0,C 180,E1 2955.947,E2 2955.947} C_VEL
LIN {X 0,Y 187.668,Z 1180.243,A -85,B 0,C 180,E1 2949.413,E2 2949.413} C_VEL
LIN {X 0,Y 191.73,Z 1176.558,A -85,B 0,C 180,E1 2943.019,E2 2943.019} C_VEL
LIN {X 0,Y 198.943,Z 1170.814,A -85,B 0,C 180,E1 2935.744,E2 2935.744} C_VEL
LIN {X 0,Y 209.137,Z 1162.956,A -85,B 0,C 180,E1 2928.718,E2 2928.718} C_VEL
LIN {X 0,Y 219.237,Z 1155.29,A -85,B 0,C 180,E1 2923.519,E2 2923.519} C_VEL
LIN {X 0,Y 232.056,Z 1145.453,A -85,B 0,C 180,E1 2918.351,E2 2918.351} C_VEL
LIN {X 0,Y 247.743,Z 1132.745,A -85,B 0,C 180,E1 2913.339,E2 2913.339} C_VEL
LIN {X 0,Y 261.462,Z 1121.003,A -85,B 0,C 180,E1 2909.764,E2 2909.764} C_VEL
LIN {X 0,Y 276.07,Z 1107.752,A -85,B 0,C 180,E1 2906.545,E2 2906.545} C_VEL
LIN {X 0,Y 293.803,Z 1090.239,A -85,B 0,C 180,E1 2903.24,E2 2903.24} C_VEL
LIN {X 0,Y 307.46,Z 1075.558,A -85,B 0,C 180,E1 2901.039,E2 2901.039} C_VEL
LIN {X 0,Y 321.17,Z 1059.645,A -85,B 0,C 180,E1 2899.08,E2 2899.08} C_VEL
LIN {X 0,Y 337.221,Z 1039.191,A -85,B 0,C 180,E1 2897.045,E2 2897.045} C_VEL
LIN {X 0,Y 350.725,Z 1019.918,A -85,B 0,C 180,E1 2895.508,E2 2895.508} C_VEL
LIN {X 0,Y 361.761,Z 1002.628,A -85,B 0,C 180,E1 2894.363,E2 2894.363} C_VEL
LIN {X 0,Y 373.171,Z 982.87,A -85,B 0,C 180,E1 2893.26,E2 2893.26} C_VEL
LIN {X 0,Y 386.014,Z 957.423,A -85,B 0,C 180,E1 2892.112,E2 2892.112} C_VEL
LIN {X 0,Y 394.722,Z 937.586,A -85,B 0,C 180,E1 2891.389,E2 2891.389} C_VEL
LIN {X 0,Y 402.083,Z 918.541,A -85,B 0,C 180,E1 2890.809,E2 2890.809} C_VEL
LIN {X 0,Y 409.476,Z 896.362,A -85,B 0,C 180,E1 2890.244,E2 2890.244} C_VEL
LIN {X 0,Y 417.11,Z 867.949,A -85,B 0,C 180,E1 2889.695,E2 2889.695} C_VEL
LIN {X 0,Y 421.795,Z 845.177,A -85,B 0,C 180,E1 2889.346,E2 2889.346} C_VEL
LIN {X 0,Y 425.361,Z 821.615,A -85,B 0,C 180,E1 2889.019,E2 2889.019} C_VEL
LIN {X 0,Y 444.791,Z 650.072,A -85,B 0,C 180,E1 2886.794,E2 2886.794} C_VEL
LIN {X 0,Y 444.156,Z 648.102,A -85,B 0,C 180,E1 2885.166,E2 2885.166} C_VEL
LIN {X 0,Y 443.733,Z 645.96,A -85,B 0,C 180,E1 2882.842,E2 2882.842} C_VEL
LIN {X 0,Y 443.751,Z 645.776,A -85,B 0,C 180,E1 2881.124,E2 2881.124} C_VEL
LIN {X 0,Y 443.733,Z 646.808,A -85,B 0,C 180,E1 2880.468,E2 2880.468} C_VEL
LIN {X 0,Y 443.433,Z 654.183,A -85,B 0,C 180,E1 2878.639,E2 2878.639} C_VEL
LIN {X 0,Y 443.523,Z 654.943,A -85,B 0,C 180,E1 2878.26,E2 2878.26} C_VEL
LIN {X 0,Y 443.772,Z 655.926,A -85,B 0,C 180,E1 2877.591,E2 2877.591} C_VEL
LIN {X 0,Y 423.776,Z 827.964,A -85,B 0,C 180,E1 2875.327,E2 2875.327} C_VEL
LIN {X 0,Y 419.219,Z 854.804,A -85,B 0,C 180,E1 2874.942,E2 2874.942} C_VEL
LIN {X 0,Y 412.937,Z 880.826,A -85,B 0,C 180,E1 2874.506,E2 2874.506} C_VEL
LIN {X 0,Y 406.684,Z 902.013,A -85,B 0,C 180,E1 2874.056,E2 2874.056} C_VEL
LIN {X 0,Y 399.028,Z 923.997,A -85,B 0,C 180,E1 2873.482,E2 2873.482} C_VEL
LIN {X 0,Y 388.157,Z 950.272,A -85,B 0,C 180,E1 2872.63,E2 2872.63} C_VEL
LIN {X 0,Y 378.1,Z 971.185,A -85,B 0,C 180,E1 2871.79,E2 2871.79} C_VEL
LIN {X 0,Y 367.624,Z 990.622,A -85,B 0,C 180,E1 2870.857,E2 2870.857} C_VEL
LIN {X 0,Y 354.359,Z 1012.739,A -85,B 0,C 180,E1 2869.571,E2 2869.571} C_VEL
LIN {X 0,Y 339.839,Z 1033.99,A -85,B 0,C 180,E1 2868.036,E2 2868.036} C_VEL
LIN {X 0,Y 327.239,Z 1050.811,A -85,B 0,C 180,E1 2866.572,E2 2866.572} C_VEL
LIN {X 0,Y 313.43,Z 1067.775,A -85,B 0,C 180,E1 2864.797,E2 2864.797} C_VEL
LIN {X 0,Y 296.054,Z 1087.316,A -85,B 0,C 180,E1 2862.252,E2 2862.252} C_VEL
LIN {X 0,Y 280.512,Z 1103.215,A -85,B 0,C 180,E1 2859.627,E2 2859.627} C_VEL
LIN {X 0,Y 266.38,Z 1116.741,A -85,B 0,C 180,E1 2856.87,E2 2856.87} C_VEL
LIN {X 0,Y 250.272,Z 1131.276,A -85,B 0,C 180,E1 2853.162,E2 2853.162} C_VEL
LIN {X 0,Y 233.506,Z 1145.334,A -85,B 0,C 180,E1 2848.442,E2 2848.442} C_VEL
LIN {X 0,Y 220.987,Z 1155.429,A -85,B 0,C 180,E1 2844.085,E2 2844.085} C_VEL
LIN {X 0,Y 209.235,Z 1164.705,A -85,B 0,C 180,E1 2839.028,E2 2839.028} C_VEL
LIN {X 0,Y 196.557,Z 1174.75,A -85,B 0,C 180,E1 2831.788,E2 2831.788} C_VEL
LIN {X 0,Y 188.127,Z 1181.648,A -85,B 0,C 180,E1 2825.03,E2 2825.03} C_VEL
LIN {X 0,Y 182.452,Z 1186.772,A -85,B 0,C 180,E1 2818.474,E2 2818.474} C_VEL
LIN {X 0,Y 178.728,Z 1190.733,A -85,B 0,C 180,E1 2811.769,E2 2811.769} C_VEL
LIN {X 0,Y 176.738,Z 1193.58,A -85,B 0,C 180,E1 2805.084,E2 2805.084} C_VEL
LIN {X 0,Y 176.069,Z 1195.388,A -85,B 0,C 180,E1 2798.49,E2 2798.49} C_VEL
LIN {X 0,Y 176.022,Z 1196.126,A -85,B 0,C 180,E1 2792.93,E2 2792.93} C_VEL
LIN {X 0,Y 176.029,Z 1196.195,A -85,B 0,C 180,E1 2788.046,E2 2788.046} C_VEL
LIN {X 0,Y 176.053,Z 1195.522,A -85,B 0,C 180,E1 2782.165,E2 2782.165} C_VEL
LIN {X 0,Y 176.678,Z 1193.681,A -85,B 0,C 180,E1 2775.245,E2 2775.245} C_VEL
LIN {X 0,Y 178.551,Z 1190.923,A -85,B 0,C 180,E1 2768.653,E2 2768.653} C_VEL
LIN {X 0,Y 182.229,Z 1186.952,A -85,B 0,C 180,E1 2761.843,E2 2761.843} C_VEL
LIN {X 0,Y 187.812,Z 1181.866,A -85,B 0,C 180,E1 2755.274,E2 2755.274} C_VEL
LIN {X 0,Y 196.139,Z 1175.007,A -85,B 0,C 180,E1 2748.492,E2 2748.492} C_VEL
LIN {X 0,Y 208.709,Z 1165.042,A -85,B 0,C 180,E1 2741.222,E2 2741.222} C_VEL
LIN {X 0,Y 220.389,Z 1155.812,A -85,B 0,C 180,E1 2736.141,E2 2736.141} C_VEL
LIN {X 0,Y 232.847,Z 1145.765,A -85,B 0,C 180,E1 2731.761,E2 2731.761} C_VEL
LIN {X 0,Y 248.589,Z 1132.63,A -85,B 0,C 180,E1 2727.263,E2 2727.263} C_VEL
LIN {X 0,Y 265.614,Z 1117.294,A -85,B 0,C 180,E1 2723.283,E2 2723.283} C_VEL
LIN {X 0,Y 279.738,Z 1103.792,A -85,B 0,C 180,E1 2720.505,E2 2720.505} C_VEL
LIN {X 0,Y 294.382,Z 1088.843,A -85,B 0,C 180,E1 2718.004,E2 2718.004} C_VEL
LIN {X 0,Y 312.643,Z 1068.467,A -85,B 0,C 180,E1 2715.302,E2 2715.302} C_VEL
LIN {X 0,Y 326.497,Z 1051.481,A -85,B 0,C 180,E1 2713.51,E2 2713.51} C_VEL
LIN {X 0,Y 338.934,Z 1034.919,A -85,B 0,C 180,E1 2712.054,E2 2712.054} C_VEL
LIN {X 0,Y 352.936,Z 1014.521,A -85,B 0,C 180,E1 2710.559,E2 2710.559} C_VEL
LIN {X 0,Y 366.967,Z 991.353,A -85,B 0,C 180,E1 2709.193,E2 2709.193} C_VEL
LIN {X 0,Y 377.372,Z 972.126,A -85,B 0,C 180,E1 2708.262,E2 2708.262} C_VEL
LIN {X 0,Y 386.739,Z 952.798,A -85,B 0,C 180,E1 2707.473,E2 2707.473} C_VEL
LIN {X 0,Y 397.163,Z 928.388,A -85,B 0,C 180,E1 2706.65,E2 2706.65} C_VEL
LIN {X 0,Y 405.917,Z 903.616,A -85,B 0,C 180,E1 2705.989,E2 2705.989} C_VEL
LIN {X 0,Y 412.426,Z 881.755,A -85,B 0,C 180,E1 2705.517,E2 2705.517} C_VEL
LIN {X 0,Y 418.208,Z 858.081,A -85,B 0,C 180,E1 2705.113,E2 2705.113} C_VEL
LIN {X 0,Y 423.317,Z 829.41,A -85,B 0,C 180,E1 2704.697,E2 2704.697} C_VEL
LIN {X 0,Y 434.032,Z 737.985,A -85,B 0,C 180,E1 2703.484,E2 2703.484} C_VEL
LIN {X 0,Y 443.544,Z 655.454,A -85,B 0,C 180,E1 2702.39,E2 2702.39} C_VEL
LIN {X 0,Y 443.002,Z 653.942,A -85,B 0,C 180,E1 2700.899,E2 2700.899} C_VEL
LIN {X 0,Y 442.476,Z 653.584,A -85,B 0,C 180,E1 2697.669,E2 2697.669} C_VEL
LIN {X 0,Y 442.567,Z 654.121,A -85,B 0,C 180,E1 2696.373,E2 2696.373} C_VEL
LIN {X 0,Y 443.1,Z 656.722,A -85,B 0,C 180,E1 2694.048,E2 2694.048} C_VEL
LIN {X 0,Y 423.173,Z 828.851,A -85,B 0,C 180,E1 2691.867,E2 2691.867} C_VEL
LIN {X 0,Y 418.586,Z 855.743,A -85,B 0,C 180,E1 2691.493,E2 2691.493} C_VEL
LIN {X 0,Y 412.507,Z 880.972,A -85,B 0,C 180,E1 2691.076,E2 2691.076} C_VEL
LIN {X 0,Y 406.346,Z 901.837,A -85,B 0,C 180,E1 2690.654,E2 2690.654} C_VEL
LIN {X 0,Y 398.264,Z 924.99,A -85,B 0,C 180,E1 2690.06,E2 2690.06} C_VEL
LIN {X 0,Y 387.766,Z 950.134,A -85,B 0,C 180,E1 2689.246,E2 2689.246} C_VEL
LIN {X 0,Y 377.979,Z 970.4,A -85,B 0,C 180,E1 2688.44,E2 2688.44} C_VEL
LIN {X 0,Y 367.623,Z 989.51,A -85,B 0,C 180,E1 2687.535,E2 2687.535} C_VEL
LIN {X 0,Y 354.114,Z 1011.828,A -85,B 0,C 180,E1 2686.246,E2 2686.246} C_VEL
LIN {X 0,Y 339.913,Z 1032.377,A -85,B 0,C 180,E1 2684.762,E2 2684.762} C_VEL
LIN {X 0,Y 327.37,Z 1048.917,A -85,B 0,C 180,E1 2683.315,E2 2683.315} C_VEL
LIN {X 0,Y 313.989,Z 1065.108,A -85,B 0,C 180,E1 2681.616,E2 2681.616} C_VEL
LIN {X 0,Y 296.048,Z 1084.81,A -85,B 0,C 180,E1 2679.022,E2 2679.022} C_VEL
LIN {X 0,Y 281.199,Z 1099.617,A -85,B 0,C 180,E1 2676.548,E2 2676.548} C_VEL
LIN {X 0,Y 267.273,Z 1112.547,A -85,B 0,C 180,E1 2673.878,E2 2673.878} C_VEL
LIN {X 0,Y 250.41,Z 1127.165,A -85,B 0,C 180,E1 2670.052,E2 2670.052} C_VEL
LIN {X 0,Y 235.19,Z 1139.285,A -85,B 0,C 180,E1 2665.862,E2 2665.862} C_VEL
LIN {X 0,Y 222.879,Z 1148.651,A -85,B 0,C 180,E1 2661.729,E2 2661.729} C_VEL
LIN {X 0,Y 210.542,Z 1157.732,A -85,B 0,C 180,E1 2656.603,E2 2656.603} C_VEL
LIN {X 0,Y 197.755,Z 1166.903,A -85,B 0,C 180,E1 2649.575,E2 2649.575} C_VEL
LIN {X 0,Y 189.489,Z 1172.91,A -85,B 0,C 180,E1 2643.284,E2 2643.284} C_VEL
LIN {X 0,Y 183.29,Z 1177.705,A -85,B 0,C 180,E1 2636.573,E2 2636.573} C_VEL
LIN {X 0,Y 178.634,Z 1181.904,A -85,B 0,C 180,E1 2628.268,E2 2628.268} C_VEL
LIN {X 0,Y 176.618,Z 1184.216,A -85,B 0,C 180,E1 2620.438,E2 2620.438} C_VEL
LIN {X 0,Y 176.11,Z 1185.175,A -85,B 0,C 180,E1 2614.233,E2 2614.233} C_VEL
LIN {X 0,Y 176.073,Z 1185.354,A -85,B 0,C 180,E1 2608.374,E2 2608.374} C_VEL
LIN {X 0,Y 176.336,Z 1184.693,A -85,B 0,C 180,E1 2601.851,E2 2601.851} C_VEL
LIN {X 0,Y 177.431,Z 1183.133,A -85,B 0,C 180,E1 2595.311,E2 2595.311} C_VEL
LIN {X 0,Y 180.048,Z 1180.495,A -85,B 0,C 180,E1 2588.499,E2 2588.499} C_VEL
LIN {X 0,Y 184.452,Z 1176.811,A -85,B 0,C 180,E1 2581.862,E2 2581.862} C_VEL
LIN {X 0,Y 192.18,Z 1171.068,A -85,B 0,C 180,E1 2574.359,E2 2574.359} C_VEL
LIN {X 0,Y 202.993,Z 1163.213,A -85,B 0,C 180,E1 2567.177,E2 2567.177} C_VEL
LIN {X 0,Y 213.626,Z 1155.55,A -85,B 0,C 180,E1 2561.91,E2 2561.91} C_VEL
LIN {X 0,Y 226.459,Z 1146.114,A -85,B 0,C 180,E1 2556.905,E2 2556.905} C_VEL
LIN {X 0,Y 243.3,Z 1133.01,A -85,B 0,C 180,E1 2551.714,E2 2551.714} C_VEL
LIN {X 0,Y 257.468,Z 1121.273,A -85,B 0,C 180,E1 2548.171,E2 2548.171} C_VEL
LIN {X 0,Y 272.494,Z 1108.026,A -85,B 0,C 180,E1 2544.998,E2 2544.998} C_VEL
LIN {X 0,Y 290.667,Z 1090.527,A -85,B 0,C 180,E1 2541.755,E2 2541.755} C_VEL
LIN {X 0,Y 305.191,Z 1075.233,A -85,B 0,C 180,E1 2539.523,E2 2539.523} C_VEL
LIN {X 0,Y 319.497,Z 1058.899,A -85,B 0,C 180,E1 2537.58,E2 2537.58} C_VEL
LIN {X 0,Y 336.285,Z 1037.668,A -85,B 0,C 180,E1 2535.561,E2 2535.561} C_VEL
LIN {X 0,Y 348.93,Z 1019.855,A -85,B 0,C 180,E1 2534.197,E2 2534.197} C_VEL
LIN {X 0,Y 360.294,Z 1002.281,A -85,B 0,C 180,E1 2533.074,E2 2533.074} C_VEL
LIN {X 0,Y 372.075,Z 982.106,A -85,B 0,C 180,E1 2531.994,E2 2531.994} C_VEL
LIN {X 0,Y 384.361,Z 958.023,A -85,B 0,C 180,E1 2530.947,E2 2530.947} C_VEL
LIN {X 0,Y 393.683,Z 937.012,A -85,B 0,C 180,E1 2530.209,E2 2530.209} C_VEL
LIN {X 0,Y 401.13,Z 917.885,A -85,B 0,C 180,E1 2529.654,E2 2529.654} C_VEL
LIN {X 0,Y 408.793,Z 895.016,A -85,B 0,C 180,E1 2529.1,E2 2529.1} C_VEL
LIN {X 0,Y 416.18,Z 867.492,A -85,B 0,C 180,E1 2528.592,E2 2528.592} C_VEL
LIN {X 0,Y 420.873,Z 844.854,A -85,B 0,C 180,E1 2528.258,E2 2528.258} C_VEL
LIN {X 0,Y 424.554,Z 820.69,A -85,B 0,C 180,E1 2527.932,E2 2527.932} C_VEL
LIN {X 0,Y 443.427,Z 656.76,A -85,B 0,C 180,E1 2525.853,E2 2525.853} C_VEL
LIN {X 0,Y 442.759,Z 653.904,A -85,B 0,C 180,E1 2522.848,E2 2522.848} C_VEL
LIN {X 0,Y 443.116,Z 654.008,A -85,B 0,C 180,E1 2519.483,E2 2519.483} C_VEL
LIN {X 0,Y 443.501,Z 654.87,A -85,B 0,C 180,E1 2518.32,E2 2518.32} C_VEL
LIN {X 0,Y 443.523,Z 654.943,A -85,B 0,C 180,E1 2518.26,E2 2518.26} C_VEL
LIN {X 0,Y 443.476,Z 656.324,A -85,B 0,C 180,E1 2518.023,E2 2518.023} C_VEL
LIN {X 0,Y 443.168,Z 659.368,A -85,B 0,C 180,E1 2517.898,E2 2517.898} C_VEL
LIN {X 0,Y 442.525,Z 664.339,A -85,B 0,C 180,E1 2517.947,E2 2517.947} C_VEL
LIN {X 0,Y 440.999,Z 675.09,A -85,B 0,C 180,E1 2518.319,E2 2518.319} C_VEL
LIN {X 0,Y 440.538,Z 678.75,A -85,B 0,C 180,E1 2518.335,E2 2518.335} C_VEL
LIN {X 0,Y 422.903,Z 828.27,A -85,B 0,C 180,E1 2516.404,E2 2516.404} C_VEL
LIN {X 0,Y 418.233,Z 855.278,A -85,B 0,C 180,E1 2516.027,E2 2516.027} C_VEL
LIN {X 0,Y 411.96,Z 880.984,A -85,B 0,C 180,E1 2515.612,E2 2515.612} C_VEL
LIN {X 0,Y 405.656,Z 902.111,A -85,B 0,C 180,E1 2515.181,E2 2515.181} C_VEL
LIN {X 0,Y 397.705,Z 924.665,A -85,B 0,C 180,E1 2514.614,E2 2514.614} C_VEL
LIN {X 0,Y 386.715,Z 950.787,A -85,B 0,C 180,E1 2513.796,E2 2513.796} C_VEL
LIN {X 0,Y 376.756,Z 971.227,A -85,B 0,C 180,E1 2513.004,E2 2513.004} C_VEL
LIN {X 0,Y 366.405,Z 990.202,A -85,B 0,C 180,E1 2512.128,E2 2512.128} C_VEL
LIN {X 0,Y 352.698,Z 1012.762,A -85,B 0,C 180,E1 2510.865,E2 2510.865} C_VEL
LIN {X 0,Y 337.76,Z 1034.263,A -85,B 0,C 180,E1 2509.363,E2 2509.363} C_VEL
LIN {X 0,Y 325.104,Z 1050.858,A -85,B 0,C 180,E1 2507.965,E2 2507.965} C_VEL
LIN {X 0,Y 310.997,Z 1067.862,A -85,B 0,C 180,E1 2506.236,E2 2506.236} C_VEL
LIN {X 0,Y 292.753,Z 1087.883,A -85,B 0,C 180,E1 2503.684,E2 2503.684} C_VEL
LIN {X 0,Y 277.697,Z 1102.927,A -85,B 0,C 180,E1 2501.253,E2 2501.253} C_VEL
LIN {X 0,Y 263.184,Z 1116.457,A -85,B 0,C 180,E1 2498.557,E2 2498.557} C_VEL
LIN {X 0,Y 247.629,Z 1130.072,A -85,B 0,C 180,E1 2495.169,E2 2495.169} C_VEL
LIN {X 0,Y 229.867,Z 1144.535,A -85,B 0,C 180,E1 2490.453,E2 2490.453} C_VEL
LIN {X 0,Y 216.423,Z 1154.937,A -85,B 0,C 180,E1 2486.011,E2 2486.011} C_VEL
LIN {X 0,Y 204.353,Z 1164.019,A -85,B 0,C 180,E1 2481.074,E2 2481.074} C_VEL
LIN {X 0,Y 191.712,Z 1173.533,A -85,B 0,C 180,E1 2474.336,E2 2474.336} C_VEL
LIN {X 0,Y 181.328,Z 1181.387,A -85,B 0,C 180,E1 2466.55,E2 2466.55} C_VEL
LIN {X 0,Y 175.18,Z 1186.514,A -85,B 0,C 180,E1 2459.772,E2 2459.772} C_VEL
LIN {X 0,Y 171.049,Z 1190.529,A -85,B 0,C 180,E1 2452.693,E2 2452.693} C_VEL
LIN {X 0,Y 168.795,Z 1193.449,A -85,B 0,C 180,E1 2445.459,E2 2445.459} C_VEL
LIN {X 0,Y 168.062,Z 1195.285,A -85,B 0,C 180,E1 2438.208,E2 2438.208} C_VEL
LIN {X 0,Y 168.032,Z 1195.951,A -85,B 0,C 180,E1 2432.045,E2 2432.045} C_VEL
LIN {X 0,Y 168.025,Z 1195.874,A -85,B 0,C 180,E1 2426.929,E2 2426.929} C_VEL
LIN {X 0,Y 168.072,Z 1195.2,A -85,B 0,C 180,E1 2421.446,E2 2421.446} C_VEL
LIN {X 0,Y 168.796,Z 1193.428,A -85,B 0,C 180,E1 2414.539,E2 2414.539} C_VEL
LIN {X 0,Y 170.943,Z 1190.617,A -85,B 0,C 180,E1 2407.547,E2 2407.547} C_VEL
LIN {X 0,Y 174.936,Z 1186.693,A -85,B 0,C 180,E1 2400.557,E2 2400.557} C_VEL
LIN {X 0,Y 180.988,Z 1181.606,A -85,B 0,C 180,E1 2393.762,E2 2393.762} C_VEL
LIN {X 0,Y 190.362,Z 1174.428,A -85,B 0,C 180,E1 2386.521,E2 2386.521} C_VEL
LIN {X 0,Y 203.41,Z 1164.647,A -85,B 0,C 180,E1 2379.355,E2 2379.355} C_VEL
LIN {X 0,Y 215.507,Z 1155.542,A -85,B 0,C 180,E1 2374.323,E2 2374.323} C_VEL
LIN {X 0,Y 228.688,Z 1145.343,A -85,B 0,C 180,E1 2369.897,E2 2369.897} C_VEL
LIN {X 0,Y 245.637,Z 1131.675,A -85,B 0,C 180,E1 2365.304,E2 2365.304} C_VEL
LIN {X 0,Y 262.386,Z 1117.015,A -85,B 0,C 180,E1 2361.593,E2 2361.593} C_VEL
LIN {X 0,Y 276.867,Z 1103.532,A -85,B 0,C 180,E1 2358.881,E2 2358.881} C_VEL
LIN {X 0,Y 291.896,Z 1088.542,A -85,B 0,C 180,E1 2356.436,E2 2356.436} C_VEL
LIN {X 0,Y 310.459,Z 1068.24,A -85,B 0,C 180,E1 2353.825,E2 2353.825} C_VEL
LIN {X 0,Y 324.514,Z 1051.314,A -85,B 0,C 180,E1 2352.094,E2 2352.094} C_VEL
LIN {X 0,Y 337.134,Z 1034.786,A -85,B 0,C 180,E1 2350.692,E2 2350.692} C_VEL
LIN {X 0,Y 351.101,Z 1014.753,A -85,B 0,C 180,E1 2349.274,E2 2349.274} C_VEL
LIN {X 0,Y 365.463,Z 991.409,A -85,B 0,C 180,E1 2347.943,E2 2347.943} C_VEL
LIN {X 0,Y 375.807,Z 972.569,A -85,B 0,C 180,E1 2347.062,E2 2347.062} C_VEL
LIN {X 0,Y 385.283,Z 953.3,A -85,B 0,C 180,E1 2346.303,E2 2346.303} C_VEL
LIN {X 0,Y 394.826,Z 931.34,A -85,B 0,C 180,E1 2345.582,E2 2345.582} C_VEL
LIN {X 0,Y 404.427,Z 905.113,A -85,B 0,C 180,E1 2344.894,E2 2344.894} C_VEL
LIN {X 0,Y 411.178,Z 882.853,A -85,B 0,C 180,E1 2344.427,E2 2344.427} C_VEL
LIN {X 0,Y 416.744,Z 860.567,A -85,B 0,C 180,E1 2344.056,E2 2344.056} C_VEL
LIN {X 0,Y 422.068,Z 832.366,A -85,B 0,C 180,E1 2343.655,E2 2343.655} C_VEL
LIN {X 0,Y 428.507,Z 779.651,A -85,B 0,C 180,E1 2342.965,E2 2342.965} C_VEL
LIN {X 0,Y 442.195,Z 662.35,A -85,B 0,C 180,E1 2341.447,E2 2341.447} C_VEL
LIN {X 0,Y 441.595,Z 661.442,A -85,B 0,C 180,E1 2339.092,E2 2339.092} C_VEL
LIN {X 0,Y 441.569,Z 661.863,A -85,B 0,C 180,E1 2336.625,E2 2336.625} C_VEL
LIN {X 0,Y 441.796,Z 663.776,A -85,B 0,C 180,E1 2334.999,E2 2334.999} C_VEL
LIN {X 0,Y 422.378,Z 828.786,A -85,B 0,C 180,E1 2332.95,E2 2332.95} C_VEL
LIN {X 0,Y 417.746,Z 855.655,A -85,B 0,C 180,E1 2332.587,E2 2332.587} C_VEL
LIN {X 0,Y 411.588,Z 880.962,A -85,B 0,C 180,E1 2332.186,E2 2332.186} C_VEL
LIN {X 0,Y 405.553,Z 901.245,A -85,B 0,C 180,E1 2331.795,E2 2331.795} C_VEL
LIN {X 0,Y 398.063,Z 922.647,A -85,B 0,C 180,E1 2331.272,E2 2331.272} C_VEL
LIN {X 0,Y 387.449,Z 948.3,A -85,B 0,C 180,E1 2330.493,E2 2330.493} C_VEL
LIN {X 0,Y 377.51,Z 968.819,A -85,B 0,C 180,E1 2329.725,E2 2329.725} C_VEL
LIN {X 0,Y 366.888,Z 988.325,A -85,B 0,C 180,E1 2328.845,E2 2328.845} C_VEL
LIN {X 0,Y 354.551,Z 1008.634,A -85,B 0,C 180,E1 2327.735,E2 2327.735} C_VEL
LIN {X 0,Y 339.217,Z 1030.92,A -85,B 0,C 180,E1 2326.226,E2 2326.226} C_VEL
LIN {X 0,Y 326.011,Z 1048.147,A -85,B 0,C 180,E1 2324.79,E2 2324.79} C_VEL
LIN {X 0,Y 312.373,Z 1064.424,A -85,B 0,C 180,E1 2323.152,E2 2323.152} C_VEL
LIN {X 0,Y 295.323,Z 1083.008,A -85,B 0,C 180,E1 2320.827,E2 2320.827} C_VEL
LIN {X 0,Y 278.841,Z 1099.144,A -85,B 0,C 180,E1 2318.239,E2 2318.239} C_VEL
LIN {X 0,Y 264.529,Z 1112.137,A -85,B 0,C 180,E1 2315.637,E2 2315.637} C_VEL
LIN {X 0,Y 247.861,Z 1126.264,A -85,B 0,C 180,E1 2312.062,E2 2312.062} C_VEL
LIN {X 0,Y 231.547,Z 1138.89,A -85,B 0,C 180,E1 2307.821,E2 2307.821} C_VEL
LIN {X 0,Y 218.477,Z 1148.469,A -85,B 0,C 180,E1 2303.657,E2 2303.657} C_VEL
LIN {X 0,Y 206.052,Z 1157.208,A -85,B 0,C 180,E1 2298.777,E2 2298.777} C_VEL
LIN {X 0,Y 192.366,Z 1166.575,A -85,B 0,C 180,E1 2291.707,E2 2291.707} C_VEL
LIN {X 0,Y 182.907,Z 1172.995,A -85,B 0,C 180,E1 2284.915,E2 2284.915} C_VEL
LIN {X 0,Y 176.246,Z 1177.763,A -85,B 0,C 180,E1 2278.092,E2 2278.092} C_VEL
LIN {X 0,Y 171.205,Z 1181.89,A -85,B 0,C 180,E1 2269.801,E2 2269.801} C_VEL
LIN {X 0,Y 168.739,Z 1184.402,A -85,B 0,C 180,E1 2261.277,E2 2261.277} C_VEL
LIN {X 0,Y 168.12,Z 1185.423,A -85,B 0,C 180,E1 2254.435,E2 2254.435} C_VEL
LIN {X 0,Y 168.077,Z 1185.601,A -85,B 0,C 180,E1 2248.296,E2 2248.296} C_VEL
